LIN {X 0,Y 424.164,Z 335.01,A -85,B 0,C 180,E1 -10008.17,E2 -10008.17} C_VEL
LIN {X 0,Y 418.479,Z 320.385,A -85,B 0,C 180,E1 -10008.722,E2 -10008.722} C_VEL
LIN {X 0,Y 418.313,Z 319.478,A -85,B 0,C 180,E1 -10008.901,E2 -10008.901} C_VEL
LIN {X 0,Y 418.234,Z 319.369,A -85,B 0,C 180,E1 -10012.448,E2 -10012.448} C_VEL
LIN {X 0,Y 418.244,Z 319.388,A -85,B 0,C 180,E1 -10014.852,E2 -10014.852} C_VEL
LIN {X 0,Y 418.201,Z 319.366,A -85,B 0,C 180,E1 -10018.069,E2 -10018.069} C_VEL
LIN {X 0,Y 418.233,Z 319.388,A -85,B 0,C 180,E1 -10021.018,E2 -10021.018} C_VEL
LIN {X 0,Y 418.25,Z 319.387,A -85,B 0,C 180,E1 -10024.577,E2 -10024.577} C_VEL
LIN {X 0,Y 418.216,Z 319.377,A -85,B 0,C 180,E1 -10027.831,E2 -10027.831} C_VEL
LIN {X 0,Y 418.204,Z 319.389,A -85,B 0,C 180,E1 -10030.949,E2 -10030.949} C_VEL
LIN {X 0,Y 418.198,Z 319.375,A -85,B 0,C 180,E1 -10033.727,E2 -10033.727} C_VEL
LIN {X 0,Y 418.195,Z 319.394,A -85,B 0,C 180,E1 -10036.447,E2 -10036.447} C_VEL
LIN {X 0,Y 418.202,Z 319.379,A -85,B 0,C 180,E1 -10039.132,E2 -10039.132} C_VEL
LIN {X 0,Y 418.231,Z 319.378,A -85,B 0,C 180,E1 -10042.775,E2 -10042.775} C_VEL
LIN {X 0,Y 418.227,Z 319.39,A -85,B 0,C 180,E1 -10046.321,E2 -10046.321} C_VEL
LIN {X 0,Y 418.232,Z 319.36,A -85,B 0,C 180,E1 -10049.727,E2 -10049.727} C_VEL
LIN {X 0,Y 418.204,Z 319.382,A -85,B 0,C 180,E1 -10053.016,E2 -10053.016} C_VEL
LIN {X 0,Y 418.248,Z 319.387,A -85,B 0,C 180,E1 -10056.216,E2 -10056.216} C_VEL
LIN {X 0,Y 418.238,Z 319.376,A -85,B 0,C 180,E1 -10059.336,E2 -10059.336} C_VEL
LIN {X 0,Y 418.266,Z 319.387,A -85,B 0,C 180,E1 -10062.395,E2 -10062.395} C_VEL
LIN {X 0,Y 418.279,Z 319.367,A -85,B 0,C 180,E1 -10065.402,E2 -10065.402} C_VEL
LIN {X 0,Y 418.303,Z 319.381,A -85,B 0,C 180,E1 -10068.369,E2 -10068.369} C_VEL
LIN {X 0,Y 418.439,Z 319.353,A -85,B 0,C 180,E1 -10072.278,E2 -10072.278} C_VEL
LIN {X 0,Y 418.456,Z 319.357,A -85,B 0,C 180,E1 -10074.216,E2 -10074.216} C_VEL
LIN {X 0,Y 418.529,Z 319.347,A -85,B 0,C 180,E1 -10078.075,E2 -10078.075} C_VEL
LIN {X 0,Y 418.463,Z 319.355,A -85,B 0,C 180,E1 -10080.962,E2 -10080.962} C_VEL
LIN {X 0,Y 418.461,Z 319.357,A -85,B 0,C 180,E1 -10082.888,E2 -10082.888} C_VEL
LIN {X 0,Y 418.49,Z 319.346,A -85,B 0,C 180,E1 -10085.783,E2 -10085.783} C_VEL
LIN {X 0,Y 418.366,Z 319.37,A -85,B 0,C 180,E1 -10088.696,E2 -10088.696} C_VEL
LIN {X 0,Y 418.346,Z 319.364,A -85,B 0,C 180,E1 -10092.615,E2 -10092.615} C_VEL
LIN {X 0,Y 418.293,Z 319.377,A -85,B 0,C 180,E1 -10095.594,E2 -10095.594} C_VEL
LIN {X 0,Y 418.267,Z 319.373,A -85,B 0,C 180,E1 -10098.618,E2 -10098.618} C_VEL
LIN {X 0,Y 418.227,Z 319.371,A -85,B 0,C 180,E1 -10101.697,E2 -10101.697} C_VEL
LIN {X 0,Y 418.238,Z 319.385,A -85,B 0,C 180,E1 -10104.853,E2 -10104.853} C_VEL
LIN {X 0,Y 418.218,Z 319.377,A -85,B 0,C 180,E1 -10108.069,E2 -10108.069} C_VEL
LIN {X 0,Y 418.205,Z 319.389,A -85,B 0,C 180,E1 -10111.397,E2 -10111.397} C_VEL
LIN {X 0,Y 418.246,Z 319.377,A -85,B 0,C 180,E1 -10114.578,E2 -10114.578} C_VEL
LIN {X 0,Y 418.211,Z 319.392,A -85,B 0,C 180,E1 -10117.832,E2 -10117.832} C_VEL
LIN {X 0,Y 418.203,Z 319.39,A -85,B 0,C 180,E1 -10120.95,E2 -10120.95} C_VEL
LIN {X 0,Y 418.198,Z 319.378,A -85,B 0,C 180,E1 -10123.729,E2 -10123.729} C_VEL
LIN {X 0,Y 418.194,Z 319.382,A -85,B 0,C 180,E1 -10126.448,E2 -10126.448} C_VEL
LIN {X 0,Y 418.203,Z 319.387,A -85,B 0,C 180,E1 -10129.134,E2 -10129.134} C_VEL
LIN {X 0,Y 418.23,Z 319.388,A -85,B 0,C 180,E1 -10132.776,E2 -10132.776} C_VEL
LIN {X 0,Y 418.23,Z 319.385,A -85,B 0,C 180,E1 -10136.322,E2 -10136.322} C_VEL
LIN {X 0,Y 418.282,Z 319.584,A -85,B 0,C 180,E1 -10137.85,E2 -10137.85} C_VEL
LIN {X 0,Y 421.611,Z 333.785,A -85,B 0,C 180,E1 -10140.357,E2 -10140.357} C_VEL
LIN {X 0,Y 422.933,Z 341.038,A -85,B 0,C 180,E1 -10141.57,E2 -10141.57} C_VEL
LIN {X 0,Y 421.685,Z 360.969,A -85,B 0,C 180,E1 -10144.586,E2 -10144.586} C_VEL
LIN {X 0,Y 420.463,Z 381.404,A -85,B 0,C 180,E1 -10147.65,E2 -10147.65} C_VEL
LIN {X 0,Y 419.398,Z 403.02,A -85,B 0,C 180,E1 -10150.874,E2 -10150.874} C_VEL
LIN {X 0,Y 423.294,Z 439.321,A -85,B 0,C 180,E1 -10151.702,E2 -10151.702} C_VEL
LIN {X 0,Y 422.516,Z 513.567,A -85,B 0,C 180,E1 -10152.984,E2 -10152.984} C_VEL
LIN {X 0,Y 422.025,Z 526.877,A -85,B 0,C 180,E1 -10153.399,E2 -10153.399} C_VEL
LIN {X 0,Y 421.283,Z 539.091,A -85,B 0,C 180,E1 -10153.961,E2 -10153.961} C_VEL
LIN {X 0,Y 420.463,Z 551.46,A -85,B 0,C 180,E1 -10154.737,E2 -10154.737} C_VEL
LIN {X 0,Y 419.557,Z 563.169,A -85,B 0,C 180,E1 -10155.696,E2 -10155.696} C_VEL
LIN {X 0,Y 418.897,Z 574.07,A -85,B 0,C 180,E1 -10156.82,E2 -10156.82} C_VEL
LIN {X 0,Y 418.543,Z 580.651,A -85,B 0,C 180,E1 -10157.638,E2 -10157.638} C_VEL
LIN {X 0,Y 417.995,Z 588.983,A -85,B 0,C 180,E1 -10158.851,E2 -10158.851} C_VEL
LIN {X 0,Y 417.634,Z 597.2,A -85,B 0,C 180,E1 -10160.312,E2 -10160.312} C_VEL
LIN {X 0,Y 417.519,Z 603.829,A -85,B 0,C 180,E1 -10161.774,E2 -10161.774} C_VEL
LIN {X 0,Y 417.47,Z 609.435,A -85,B 0,C 180,E1 -10163.34,E2 -10163.34} C_VEL
LIN {X 0,Y 417.644,Z 614.342,A -85,B 0,C 180,E1 -10165.174,E2 -10165.174} C_VEL
LIN {X 0,Y 417.711,Z 616.278,A -85,B 0,C 180,E1 -10166.141,E2 -10166.141} C_VEL
LIN {X 0,Y 417.687,Z 617.72,A -85,B 0,C 180,E1 -10167.107,E2 -10167.107} C_VEL
LIN {X 0,Y 417.947,Z 619.416,A -85,B 0,C 180,E1 -10169.037,E2 -10169.037} C_VEL
LIN {X 0,Y 417.96,Z 619.641,A -85,B 0,C 180,E1 -10170,E2 -10170} C_VEL
LIN {X 0,Y 417.947,Z 619.415,A -85,B 0,C 180,E1 -10170.963,E2 -10170.963} C_VEL
LIN {X 0,Y 417.688,Z 617.719,A -85,B 0,C 180,E1 -10172.893,E2 -10172.893} C_VEL
LIN {X 0,Y 417.711,Z 616.275,A -85,B 0,C 180,E1 -10173.859,E2 -10173.859} C_VEL
LIN {X 0,Y 417.551,Z 613.215,A -85,B 0,C 180,E1 -10175.312,E2 -10175.312} C_VEL
LIN {X 0,Y 417.519,Z 609.099,A -85,B 0,C 180,E1 -10176.767,E2 -10176.767} C_VEL
LIN {X 0,Y 417.519,Z 602.781,A -85,B 0,C 180,E1 -10178.47,E2 -10178.47} C_VEL
LIN {X 0,Y 417.664,Z 595.91,A -85,B 0,C 180,E1 -10179.932,E2 -10179.932} C_VEL
LIN {X 0,Y 418.089,Z 587.435,A -85,B 0,C 180,E1 -10181.391,E2 -10181.391} C_VEL
LIN {X 0,Y 418.703,Z 578.787,A -85,B 0,C 180,E1 -10182.604,E2 -10182.604} C_VEL
LIN {X 0,Y 419.221,Z 569.303,A -85,B 0,C 180,E1 -10183.697,E2 -10183.697} C_VEL
LIN {X 0,Y 419.925,Z 557.585,A -85,B 0,C 180,E1 -10184.787,E2 -10184.787} C_VEL
LIN {X 0,Y 420.82,Z 546.111,A -85,B 0,C 180,E1 -10185.622,E2 -10185.622} C_VEL
LIN {X 0,Y 421.537,Z 534.336,A -85,B 0,C 180,E1 -10186.278,E2 -10186.278} C_VEL
LIN {X 0,Y 422.248,Z 521.736,A -85,B 0,C 180,E1 -10186.778,E2 -10186.778} C_VEL
LIN {X 0,Y 422.652,Z 508.962,A -85,B 0,C 180,E1 -10187.104,E2 -10187.104} C_VEL
LIN {X 0,Y 423.252,Z 438.649,A -85,B 0,C 180,E1 -10188.305,E2 -10188.305} C_VEL
LIN {X 0,Y 419.395,Z 403.264,A -85,B 0,C 180,E1 -10189.104,E2 -10189.104} C_VEL
LIN {X 0,Y 419.602,Z 397.115,A -85,B 0,C 180,E1 -10189.982,E2 -10189.982} C_VEL
LIN {X 0,Y 420.761,Z 376.002,A -85,B 0,C 180,E1 -10193.15,E2 -10193.15} C_VEL
LIN {X 0,Y 422.195,Z 352.327,A -85,B 0,C 180,E1 -10196.708,E2 -10196.708} C_VEL
LIN {X 0,Y 422.873,Z 340.757,A -85,B 0,C 180,E1 -10198.467,E2 -10198.467} C_VEL
LIN {X 0,Y 420.636,Z 329.564,A -85,B 0,C 180,E1 -10200.358,E2 -10200.358} C_VEL
LIN {X 0,Y 418.275,Z 319.506,A -85,B 0,C 180,E1 -10202.169,E2 -10202.169} C_VEL
LIN {X 0,Y 418.247,Z 319.383,A -85,B 0,C 180,E1 -10204.841,E2 -10204.841} C_VEL
LIN {X 0,Y 418.231,Z 319.382,A -85,B 0,C 180,E1 -10208.443,E2 -10208.443} C_VEL
LIN {X 0,Y 418.215,Z 319.392,A -85,B 0,C 180,E1 -10212.235,E2 -10212.235} C_VEL
LIN {X 0,Y 418.23,Z 319.362,A -85,B 0,C 180,E1 -10215.108,E2 -10215.108} C_VEL
LIN {X 0,Y 418.216,Z 319.389,A -85,B 0,C 180,E1 -10217.764,E2 -10217.764} C_VEL
LIN {X 0,Y 418.228,Z 319.36,A -85,B 0,C 180,E1 -10221.555,E2 -10221.555} C_VEL
LIN {X 0,Y 418.244,Z 319.368,A -85,B 0,C 180,E1 -10225.157,E2 -10225.157} C_VEL
LIN {X 0,Y 418.238,Z 319.385,A -85,B 0,C 180,E1 -10227.471,E2 -10227.471} C_VEL
LIN {X 0,Y 418.257,Z 319.372,A -85,B 0,C 180,E1 -10230.896,E2 -10230.896} C_VEL
LIN {X 0,Y 418.224,Z 319.391,A -85,B 0,C 180,E1 -10234.093,E2 -10234.093} C_VEL
LIN {X 0,Y 418.221,Z 319.384,A -85,B 0,C 180,E1 -10237.263,E2 -10237.263} C_VEL
LIN {X 0,Y 418.276,Z 319.371,A -85,B 0,C 180,E1 -10240.364,E2 -10240.364} C_VEL
LIN {X 0,Y 418.309,Z 319.377,A -85,B 0,C 180,E1 -10243.404,E2 -10243.404} C_VEL
LIN {X 0,Y 418.339,Z 319.362,A -85,B 0,C 180,E1 -10246.999,E2 -10246.999} C_VEL
LIN {X 0,Y 418.327,Z 319.374,A -85,B 0,C 180,E1 -10250.328,E2 -10250.328} C_VEL
LIN {X 0,Y 418.458,Z 319.353,A -85,B 0,C 180,E1 -10253.248,E2 -10253.248} C_VEL
LIN {X 0,Y 418.313,Z 319.369,A -85,B 0,C 180,E1 -10255.181,E2 -10255.181} C_VEL
LIN {X 0,Y 418.524,Z 319.349,A -85,B 0,C 180,E1 -10258.075,E2 -10258.075} C_VEL
LIN {X 0,Y 418.398,Z 319.353,A -85,B 0,C 180,E1 -10260.963,E2 -10260.963} C_VEL
LIN {X 0,Y 418.473,Z 319.352,A -85,B 0,C 180,E1 -10262.888,E2 -10262.888} C_VEL
LIN {X 0,Y 418.434,Z 319.354,A -85,B 0,C 180,E1 -10266.752,E2 -10266.752} C_VEL
LIN {X 0,Y 418.329,Z 319.373,A -85,B 0,C 180,E1 -10269.672,E2 -10269.672} C_VEL
LIN {X 0,Y 418.339,Z 319.37,A -85,B 0,C 180,E1 -10273.001,E2 -10273.001} C_VEL
LIN {X 0,Y 418.304,Z 319.374,A -85,B 0,C 180,E1 -10276.735,E2 -10276.735} C_VEL
LIN {X 0,Y 418.263,Z 319.377,A -85,B 0,C 180,E1 -10279.79,E2 -10279.79} C_VEL
LIN {X 0,Y 418.221,Z 319.384,A -85,B 0,C 180,E1 -10282.737,E2 -10282.737} C_VEL
LIN {X 0,Y 418.212,Z 319.383,A -85,B 0,C 180,E1 -10285.908,E2 -10285.908} C_VEL
LIN {X 0,Y 418.25,Z 319.355,A -85,B 0,C 180,E1 -10289.163,E2 -10289.163} C_VEL
LIN {X 0,Y 418.246,Z 319.378,A -85,B 0,C 180,E1 -10292.843,E2 -10292.843} C_VEL
LIN {X 0,Y 418.238,Z 319.381,A -85,B 0,C 180,E1 -10296.238,E2 -10296.238} C_VEL
LIN {X 0,Y 418.194,Z 319.371,A -85,B 0,C 180,E1 -10299.689,E2 -10299.689} C_VEL
LIN {X 0,Y 418.203,Z 319.388,A -85,B 0,C 180,E1 -10302.318,E2 -10302.318} C_VEL
LIN {X 0,Y 418.232,Z 319.384,A -85,B 0,C 180,E1 -10305.109,E2 -10305.109} C_VEL
LIN {X 0,Y 418.214,Z 319.379,A -85,B 0,C 180,E1 -10307.765,E2 -10307.765} C_VEL
LIN {X 0,Y 418.233,Z 319.38,A -85,B 0,C 180,E1 -10311.557,E2 -10311.557} C_VEL
LIN {X 0,Y 418.249,Z 319.388,A -85,B 0,C 180,E1 -10315.159,E2 -10315.159} C_VEL
LIN {X 0,Y 418.237,Z 319.38,A -85,B 0,C 180,E1 -10317.472,E2 -10317.472} C_VEL
LIN {X 0,Y 418.258,Z 319.376,A -85,B 0,C 180,E1 -10320.899,E2 -10320.899} C_VEL
LIN {X 0,Y 418.21,Z 319.379,A -85,B 0,C 180,E1 -10324.092,E2 -10324.092} C_VEL
LIN {X 0,Y 418.227,Z 319.373,A -85,B 0,C 180,E1 -10327.264,E2 -10327.264} C_VEL
LIN {X 0,Y 418.312,Z 319.345,A -85,B 0,C 180,E1 -10330.876,E2 -10330.876} C_VEL
LIN {X 0,Y 418.37,Z 319.77,A -85,B 0,C 180,E1 -10331.292,E2 -10331.292} C_VEL
LIN {X 0,Y 418.751,Z 321.14,A -85,B 0,C 180,E1 -10331.419,E2 -10331.419} C_VEL
LIN {X 0,Y 424.249,Z 335.165,A -85,B 0,C 180,E1 -10331.934,E2 -10331.934} C_VEL
LIN {X 0,Y 423.684,Z 400.146,A -85,B 0,C 180,E1 -10333.063,E2 -10333.063} C_VEL
LIN {X 0,Y 423.564,Z 412.838,A -85,B 0,C 180,E1 -10333.461,E2 -10333.461} C_VEL
LIN {X 0,Y 423.267,Z 425.198,A -85,B 0,C 180,E1 -10334.038,E2 -10334.038} C_VEL
LIN {X 0,Y 422.856,Z 437.548,A -85,B 0,C 180,E1 -10334.824,E2 -10334.824} C_VEL
LIN {X 0,Y 422.141,Z 449.13,A -85,B 0,C 180,E1 -10335.785,E2 -10335.785} C_VEL
LIN {X 0,Y 421.492,Z 459.468,A -85,B 0,C 180,E1 -10336.869,E2 -10336.869} C_VEL
LIN {X 0,Y 420.95,Z 467.894,A -85,B 0,C 180,E1 -10337.954,E2 -10337.954} C_VEL
LIN {X 0,Y 420.346,Z 475.653,A -85,B 0,C 180,E1 -10339.159,E2 -10339.159} C_VEL
LIN {X 0,Y 419.765,Z 483.331,A -85,B 0,C 180,E1 -10340.629,E2 -10340.629} C_VEL
LIN {X 0,Y 419.323,Z 489.087,A -85,B 0,C 180,E1 -10342.002,E2 -10342.002} C_VEL
LIN {X 0,Y 419.063,Z 493.36,A -85,B 0,C 180,E1 -10343.258,E2 -10343.258} C_VEL
LIN {X 0,Y 418.611,Z 497.256,A -85,B 0,C 180,E1 -10344.702,E2 -10344.702} C_VEL
LIN {X 0,Y 418.384,Z 499.239,A -85,B 0,C 180,E1 -10345.678,E2 -10345.678} C_VEL
LIN {X 0,Y 417.623,Z 500.71,A -85,B 0,C 180,E1 -10346.457,E2 -10346.457} C_VEL
LIN {X 0,Y 414.712,Z 502.691,A -85,B 0,C 180,E1 -10347.733,E2 -10347.733} C_VEL
LIN {X 0,Y 412.317,Z 503.759,A -85,B 0,C 180,E1 -10348.773,E2 -10348.773} C_VEL
LIN {X 0,Y 411.309,Z 504.179,A -85,B 0,C 180,E1 -10349.583,E2 -10349.583} C_VEL
LIN {X 0,Y 411.235,Z 504.22,A -85,B 0,C 180,E1 -10349.857,E2 -10349.857} C_VEL
LIN {X 0,Y 411.257,Z 504.07,A -85,B 0,C 180,E1 -10350.979,E2 -10350.979} C_VEL
LIN {X 0,Y 411.181,Z 503.516,A -85,B 0,C 180,E1 -10351.959,E2 -10351.959} C_VEL
LIN {X 0,Y 411.332,Z 502.561,A -85,B 0,C 180,E1 -10352.938,E2 -10352.938} C_VEL
LIN {X 0,Y 411.294,Z 501.258,A -85,B 0,C 180,E1 -10353.919,E2 -10353.919} C_VEL
LIN {X 0,Y 411.607,Z 498.444,A -85,B 0,C 180,E1 -10355.388,E2 -10355.388} C_VEL
LIN {X 0,Y 412.065,Z 494.62,A -85,B 0,C 180,E1 -10356.857,E2 -10356.857} C_VEL
LIN {X 0,Y 412.366,Z 489.544,A -85,B 0,C 180,E1 -10358.379,E2 -10358.379} C_VEL
LIN {X 0,Y 413.052,Z 482.312,A -85,B 0,C 180,E1 -10360.044,E2 -10360.044} C_VEL
LIN {X 0,Y 413.751,Z 474.285,A -85,B 0,C 180,E1 -10361.513,E2 -10361.513} C_VEL
LIN {X 0,Y 414.321,Z 466.066,A -85,B 0,C 180,E1 -10362.739,E2 -10362.739} C_VEL
LIN {X 0,Y 414.933,Z 457.038,A -85,B 0,C 180,E1 -10363.842,E2 -10363.842} C_VEL
LIN {X 0,Y 415.695,Z 446.536,A -85,B 0,C 180,E1 -10364.872,E2 -10364.872} C_VEL
LIN {X 0,Y 416.207,Z 434.882,A -85,B 0,C 180,E1 -10365.787,E2 -10365.787} C_VEL
LIN {X 0,Y 416.655,Z 423.452,A -85,B 0,C 180,E1 -10366.474,E2 -10366.474} C_VEL
LIN {X 0,Y 416.858,Z 410.602,A -85,B 0,C 180,E1 -10367.033,E2 -10367.033} C_VEL
LIN {X 0,Y 416.904,Z 396.844,A -85,B 0,C 180,E1 -10367.411,E2 -10367.411} C_VEL
LIN {X 0,Y 417.432,Z 336.493,A -85,B 0,C 180,E1 -10368.464,E2 -10368.464} C_VEL
LIN {X 0,Y 411.427,Z 321.136,A -85,B 0,C 180,E1 -10369.068,E2 -10369.068} C_VEL
LIN {X 0,Y 411.278,Z 320.312,A -85,B 0,C 180,E1 -10369.27,E2 -10369.27} C_VEL
LIN {X 0,Y 411.187,Z 320.251,A -85,B 0,C 180,E1 -10373.148,E2 -10373.148} C_VEL
LIN {X 0,Y 411.163,Z 320.246,A -85,B 0,C 180,E1 -10376.386,E2 -10376.386} C_VEL
LIN {X 0,Y 411.193,Z 320.261,A -85,B 0,C 180,E1 -10379.713,E2 -10379.713} C_VEL
LIN {X 0,Y 411.201,Z 320.258,A -85,B 0,C 180,E1 -10383.156,E2 -10383.156} C_VEL
LIN {X 0,Y 411.188,Z 320.257,A -85,B 0,C 180,E1 -10386.551,E2 -10386.551} C_VEL
LIN {X 0,Y 411.166,Z 320.266,A -85,B 0,C 180,E1 -10389.719,E2 -10389.719} C_VEL
LIN {X 0,Y 411.158,Z 320.251,A -85,B 0,C 180,E1 -10393.135,E2 -10393.135} C_VEL
LIN {X 0,Y 411.16,Z 320.266,A -85,B 0,C 180,E1 -10395.881,E2 -10395.881} C_VEL
LIN {X 0,Y 411.153,Z 320.255,A -85,B 0,C 180,E1 -10399.492,E2 -10399.492} C_VEL
LIN {X 0,Y 411.179,Z 320.246,A -85,B 0,C 180,E1 -10402.024,E2 -10402.024} C_VEL
LIN {X 0,Y 411.197,Z 320.263,A -85,B 0,C 180,E1 -10405.123,E2 -10405.123} C_VEL
LIN {X 0,Y 411.158,Z 320.26,A -85,B 0,C 180,E1 -10408.002,E2 -10408.002} C_VEL
LIN {X 0,Y 411.165,Z 320.241,A -85,B 0,C 180,E1 -10411.406,E2 -10411.406} C_VEL
LIN {X 0,Y 411.182,Z 320.266,A -85,B 0,C 180,E1 -10414.941,E2 -10414.941} C_VEL
LIN {X 0,Y 411.194,Z 320.26,A -85,B 0,C 180,E1 -10417.913,E2 -10417.913} C_VEL
LIN {X 0,Y 411.21,Z 320.261,A -85,B 0,C 180,E1 -10421.051,E2 -10421.051} C_VEL
LIN {X 0,Y 411.236,Z 320.257,A -85,B 0,C 180,E1 -10424.131,E2 -10424.131} C_VEL
LIN {X 0,Y 411.296,Z 320.247,A -85,B 0,C 180,E1 -10427.165,E2 -10427.165} C_VEL
LIN {X 0,Y 411.273,Z 320.255,A -85,B 0,C 180,E1 -10430.161,E2 -10430.161} C_VEL
LIN {X 0,Y 411.378,Z 320.234,A -85,B 0,C 180,E1 -10433.132,E2 -10433.132} C_VEL
LIN {X 0,Y 411.28,Z 320.252,A -85,B 0,C 180,E1 -10435.099,E2 -10435.099} C_VEL
LIN {X 0,Y 411.498,Z 320.223,A -85,B 0,C 180,E1 -10438.042,E2 -10438.042} C_VEL
LIN {X 0,Y 411.493,Z 320.225,A -85,B 0,C 180,E1 -10441.957,E2 -10441.957} C_VEL
LIN {X 0,Y 411.436,Z 320.225,A -85,B 0,C 180,E1 -10445.883,E2 -10445.883} C_VEL
LIN {X 0,Y 411.406,Z 320.232,A -85,B 0,C 180,E1 -10447.855,E2 -10447.855} C_VEL
LIN {X 0,Y 411.266,Z 320.251,A -85,B 0,C 180,E1 -10451.833,E2 -10451.833} C_VEL
LIN {X 0,Y 411.251,Z 320.255,A -85,B 0,C 180,E1 -10454.853,E2 -10454.853} C_VEL
LIN {X 0,Y 411.237,Z 320.259,A -85,B 0,C 180,E1 -10457.916,E2 -10457.916} C_VEL
LIN {X 0,Y 411.189,Z 320.246,A -85,B 0,C 180,E1 -10461.035,E2 -10461.035} C_VEL
LIN {X 0,Y 411.186,Z 320.268,A -85,B 0,C 180,E1 -10464.218,E2 -10464.218} C_VEL
LIN {X 0,Y 411.175,Z 320.258,A -85,B 0,C 180,E1 -10467.484,E2 -10467.484} C_VEL
LIN {X 0,Y 411.192,Z 320.255,A -85,B 0,C 180,E1 -10469.713,E2 -10469.713} C_VEL
LIN {X 0,Y 411.199,Z 320.259,A -85,B 0,C 180,E1 -10473.157,E2 -10473.157} C_VEL
LIN {X 0,Y 411.183,Z 320.266,A -85,B 0,C 180,E1 -10476.552,E2 -10476.552} C_VEL
LIN {X 0,Y 411.163,Z 320.261,A -85,B 0,C 180,E1 -10479.721,E2 -10479.721} C_VEL
LIN {X 0,Y 411.159,Z 320.262,A -85,B 0,C 180,E1 -10483.136,E2 -10483.136} C_VEL
LIN {X 0,Y 411.158,Z 320.248,A -85,B 0,C 180,E1 -10485.883,E2 -10485.883} C_VEL
LIN {X 0,Y 411.143,Z 320.267,A -85,B 0,C 180,E1 -10488.775,E2 -10488.775} C_VEL
LIN {X 0,Y 411.178,Z 320.266,A -85,B 0,C 180,E1 -10492.025,E2 -10492.025} C_VEL
LIN {X 0,Y 411.199,Z 320.259,A -85,B 0,C 180,E1 -10495.124,E2 -10495.124} C_VEL
LIN {X 0,Y 411.231,Z 320.494,A -85,B 0,C 180,E1 -10497.539,E2 -10497.539} C_VEL
LIN {X 0,Y 414.675,Z 335.185,A -85,B 0,C 180,E1 -10500.187,E2 -10500.187} C_VEL
LIN {X 0,Y 416.05,Z 342.591,A -85,B 0,C 180,E1 -10501.45,E2 -10501.45} C_VEL
LIN {X 0,Y 414.782,Z 361.752,A -85,B 0,C 180,E1 -10504.402,E2 -10504.402} C_VEL
LIN {X 0,Y 413.494,Z 382.134,A -85,B 0,C 180,E1 -10507.517,E2 -10507.517} C_VEL
LIN {X 0,Y 412.436,Z 401.9,A -85,B 0,C 180,E1 -10510.529,E2 -10510.529} C_VEL
LIN {X 0,Y 415.827,Z 433.041,A -85,B 0,C 180,E1 -10511.269,E2 -10511.269} C_VEL
LIN {X 0,Y 416.533,Z 441.796,A -85,B 0,C 180,E1 -10511.456,E2 -10511.456} C_VEL
LIN {X 0,Y 415.691,Z 512.586,A -85,B 0,C 180,E1 -10512.696,E2 -10512.696} C_VEL
LIN {X 0,Y 415.186,Z 525.891,A -85,B 0,C 180,E1 -10513.118,E2 -10513.118} C_VEL
LIN {X 0,Y 414.433,Z 538.104,A -85,B 0,C 180,E1 -10513.688,E2 -10513.688} C_VEL
LIN {X 0,Y 413.726,Z 548.767,A -85,B 0,C 180,E1 -10514.356,E2 -10514.356} C_VEL
LIN {X 0,Y 412.815,Z 559.534,A -85,B 0,C 180,E1 -10515.205,E2 -10515.205} C_VEL
LIN {X 0,Y 412.178,Z 569.513,A -85,B 0,C 180,E1 -10516.19,E2 -10516.19} C_VEL
LIN {X 0,Y 411.592,Z 579.662,A -85,B 0,C 180,E1 -10517.426,E2 -10517.426} C_VEL
LIN {X 0,Y 410.97,Z 587.989,A -85,B 0,C 180,E1 -10518.658,E2 -10518.658} C_VEL
LIN {X 0,Y 410.555,Z 596.202,A -85,B 0,C 180,E1 -10520.144,E2 -10520.144} C_VEL
LIN {X 0,Y 410.441,Z 602.835,A -85,B 0,C 180,E1 -10521.631,E2 -10521.631} C_VEL
LIN {X 0,Y 410.419,Z 608.703,A -85,B 0,C 180,E1 -10523.31,E2 -10523.31} C_VEL
LIN {X 0,Y 410.567,Z 613.354,A -85,B 0,C 180,E1 -10525.09,E2 -10525.09} C_VEL
LIN {X 0,Y 410.669,Z 615.296,A -85,B 0,C 180,E1 -10526.075,E2 -10526.075} C_VEL
LIN {X 0,Y 410.642,Z 616.738,A -85,B 0,C 180,E1 -10527.057,E2 -10527.057} C_VEL
LIN {X 0,Y 410.918,Z 618.438,A -85,B 0,C 180,E1 -10529.02,E2 -10529.02} C_VEL
LIN {X 0,Y 410.935,Z 618.663,A -85,B 0,C 180,E1 -10530,E2 -10530} C_VEL
LIN {X 0,Y 410.918,Z 618.436,A -85,B 0,C 180,E1 -10530.98,E2 -10530.98} C_VEL
LIN {X 0,Y 410.642,Z 616.737,A -85,B 0,C 180,E1 -10532.943,E2 -10532.943} C_VEL
LIN {X 0,Y 410.67,Z 615.292,A -85,B 0,C 180,E1 -10533.925,E2 -10533.925} C_VEL
LIN {X 0,Y 410.48,Z 612.226,A -85,B 0,C 180,E1 -10535.403,E2 -10535.403} C_VEL
LIN {X 0,Y 410.434,Z 608.105,A -85,B 0,C 180,E1 -10536.884,E2 -10536.884} C_VEL
LIN {X 0,Y 410.451,Z 601.785,A -85,B 0,C 180,E1 -10538.616,E2 -10538.616} C_VEL
LIN {X 0,Y 410.609,Z 594.911,A -85,B 0,C 180,E1 -10540.104,E2 -10540.104} C_VEL
LIN {X 0,Y 411.046,Z 586.433,A -85,B 0,C 180,E1 -10541.589,E2 -10541.589} C_VEL
LIN {X 0,Y 411.701,Z 577.786,A -85,B 0,C 180,E1 -10542.821,E2 -10542.821} C_VEL
LIN {X 0,Y 412.347,Z 567.111,A -85,B 0,C 180,E1 -10544.056,E2 -10544.056} C_VEL
LIN {X 0,Y 413.032,Z 556.589,A -85,B 0,C 180,E1 -10545.039,E2 -10545.039} C_VEL
LIN {X 0,Y 413.927,Z 545.11,A -85,B 0,C 180,E1 -10545.889,E2 -10545.889} C_VEL
LIN {X 0,Y 414.729,Z 533.341,A -85,B 0,C 180,E1 -10546.553,E2 -10546.553} C_VEL
LIN {X 0,Y 415.483,Z 519.818,A -85,B 0,C 180,E1 -10547.091,E2 -10547.091} C_VEL
LIN {X 0,Y 415.838,Z 506.408,A -85,B 0,C 180,E1 -10547.425,E2 -10547.425} C_VEL
LIN {X 0,Y 416.42,Z 438.976,A -85,B 0,C 180,E1 -10548.592,E2 -10548.592} C_VEL
LIN {X 0,Y 412.45,Z 402.247,A -85,B 0,C 180,E1 -10549.438,E2 -10549.438} C_VEL
LIN {X 0,Y 412.825,Z 393.906,A -85,B 0,C 180,E1 -10550.672,E2 -10550.672} C_VEL
LIN {X 0,Y 414.078,Z 371.9,A -85,B 0,C 180,E1 -10554.038,E2 -10554.038} C_VEL
LIN {X 0,Y 415.439,Z 351.412,A -85,B 0,C 180,E1 -10557.178,E2 -10557.178} C_VEL
LIN {X 0,Y 415.988,Z 342.084,A -85,B 0,C 180,E1 -10558.625,E2 -10558.625} C_VEL
LIN {X 0,Y 413.593,Z 330.359,A -85,B 0,C 180,E1 -10560.648,E2 -10560.648} C_VEL
LIN {X 0,Y 411.235,Z 320.374,A -85,B 0,C 180,E1 -10562.497,E2 -10562.497} C_VEL
LIN {X 0,Y 411.173,Z 320.258,A -85,B 0,C 180,E1 -10565.53,E2 -10565.53} C_VEL
LIN {X 0,Y 411.174,Z 320.254,A -85,B 0,C 180,E1 -10569.228,E2 -10569.228} C_VEL
LIN {X 0,Y 411.162,Z 320.266,A -85,B 0,C 180,E1 -10572.693,E2 -10572.693} C_VEL
LIN {X 0,Y 411.159,Z 320.248,A -85,B 0,C 180,E1 -10575.881,E2 -10575.881} C_VEL
LIN {X 0,Y 411.143,Z 320.27,A -85,B 0,C 180,E1 -10578.774,E2 -10578.774} C_VEL
LIN {X 0,Y 411.176,Z 320.228,A -85,B 0,C 180,E1 -10582.024,E2 -10582.024} C_VEL
LIN {X 0,Y 411.196,Z 320.245,A -85,B 0,C 180,E1 -10585.123,E2 -10585.123} C_VEL
LIN {X 0,Y 411.158,Z 320.272,A -85,B 0,C 180,E1 -10588.002,E2 -10588.002} C_VEL
LIN {X 0,Y 411.187,Z 320.252,A -85,B 0,C 180,E1 -10591.407,E2 -10591.407} C_VEL
LIN {X 0,Y 411.206,Z 320.261,A -85,B 0,C 180,E1 -10594.933,E2 -10594.933} C_VEL
LIN {X 0,Y 411.197,Z 320.25,A -85,B 0,C 180,E1 -10597.913,E2 -10597.913} C_VEL
LIN {X 0,Y 411.215,Z 320.249,A -85,B 0,C 180,E1 -10601.051,E2 -10601.051} C_VEL
LIN {X 0,Y 411.246,Z 320.257,A -85,B 0,C 180,E1 -10604.131,E2 -10604.131} C_VEL
LIN {X 0,Y 411.296,Z 320.24,A -85,B 0,C 180,E1 -10607.165,E2 -10607.165} C_VEL
LIN {X 0,Y 411.28,Z 320.254,A -85,B 0,C 180,E1 -10610.161,E2 -10610.161} C_VEL
LIN {X 0,Y 411.424,Z 320.228,A -85,B 0,C 180,E1 -10613.132,E2 -10613.132} C_VEL
LIN {X 0,Y 411.286,Z 320.244,A -85,B 0,C 180,E1 -10615.099,E2 -10615.099} C_VEL
LIN {X 0,Y 411.493,Z 320.226,A -85,B 0,C 180,E1 -10618.043,E2 -10618.043} C_VEL
LIN {X 0,Y 411.369,Z 320.228,A -85,B 0,C 180,E1 -10620.979,E2 -10620.979} C_VEL
LIN {X 0,Y 411.431,Z 320.229,A -85,B 0,C 180,E1 -10622.937,E2 -10622.937} C_VEL
LIN {X 0,Y 411.383,Z 320.232,A -85,B 0,C 180,E1 -10626.868,E2 -10626.868} C_VEL
LIN {X 0,Y 411.282,Z 320.254,A -85,B 0,C 180,E1 -10629.839,E2 -10629.839} C_VEL
LIN {X 0,Y 411.299,Z 320.247,A -85,B 0,C 180,E1 -10633.104,E2 -10633.104} C_VEL
LIN {X 0,Y 411.251,Z 320.253,A -85,B 0,C 180,E1 -10636.889,E2 -10636.889} C_VEL
LIN {X 0,Y 411.225,Z 320.252,A -85,B 0,C 180,E1 -10639.987,E2 -10639.987} C_VEL
LIN {X 0,Y 411.182,Z 320.263,A -85,B 0,C 180,E1 -10643.149,E2 -10643.149} C_VEL
LIN {X 0,Y 411.165,Z 320.258,A -85,B 0,C 180,E1 -10646.386,E2 -10646.386} C_VEL
LIN {X 0,Y 411.189,Z 320.232,A -85,B 0,C 180,E1 -10649.714,E2 -10649.714} C_VEL
LIN {X 0,Y 411.199,Z 320.258,A -85,B 0,C 180,E1 -10653.157,E2 -10653.157} C_VEL
LIN {X 0,Y 411.186,Z 320.259,A -85,B 0,C 180,E1 -10656.553,E2 -10656.553} C_VEL
LIN {X 0,Y 411.163,Z 320.246,A -85,B 0,C 180,E1 -10659.721,E2 -10659.721} C_VEL
LIN {X 0,Y 411.159,Z 320.27,A -85,B 0,C 180,E1 -10663.136,E2 -10663.136} C_VEL
LIN {X 0,Y 411.16,Z 320.253,A -85,B 0,C 180,E1 -10665.883,E2 -10665.883} C_VEL
LIN {X 0,Y 411.155,Z 320.272,A -85,B 0,C 180,E1 -10669.494,E2 -10669.494} C_VEL
LIN {X 0,Y 411.18,Z 320.254,A -85,B 0,C 180,E1 -10672.026,E2 -10672.026} C_VEL
LIN {X 0,Y 411.201,Z 320.265,A -85,B 0,C 180,E1 -10675.124,E2 -10675.124} C_VEL
LIN {X 0,Y 411.158,Z 320.264,A -85,B 0,C 180,E1 -10678.003,E2 -10678.003} C_VEL
LIN {X 0,Y 411.168,Z 320.249,A -85,B 0,C 180,E1 -10681.407,E2 -10681.407} C_VEL
LIN {X 0,Y 411.187,Z 320.266,A -85,B 0,C 180,E1 -10684.942,E2 -10684.942} C_VEL
LIN {X 0,Y 411.203,Z 320.246,A -85,B 0,C 180,E1 -10687.914,E2 -10687.914} C_VEL
LIN {X 0,Y 411.298,Z 320.359,A -85,B 0,C 180,E1 -10690.861,E2 -10690.861} C_VEL
LIN {X 0,Y 411.44,Z 321.123,A -85,B 0,C 180,E1 -10691.03,E2 -10691.03} C_VEL
LIN {X 0,Y 417.409,Z 336.438,A -85,B 0,C 180,E1 -10691.632,E2 -10691.632} C_VEL
LIN {X 0,Y 416.955,Z 401.145,A -85,B 0,C 180,E1 -10692.781,E2 -10692.781} C_VEL
LIN {X 0,Y 416.815,Z 413.829,A -85,B 0,C 180,E1 -10693.186,E2 -10693.186} C_VEL
LIN {X 0,Y 416.511,Z 426.184,A -85,B 0,C 180,E1 -10693.772,E2 -10693.772} C_VEL
LIN {X 0,Y 416.078,Z 438.531,A -85,B 0,C 180,E1 -10694.57,E2 -10694.57} C_VEL
LIN {X 0,Y 415.329,Z 450.113,A -85,B 0,C 180,E1 -10695.547,E2 -10695.547} C_VEL
LIN {X 0,Y 414.649,Z 460.45,A -85,B 0,C 180,E1 -10696.648,E2 -10696.648} C_VEL
LIN {X 0,Y 414.078,Z 468.876,A -85,B 0,C 180,E1 -10697.751,E2 -10697.751} C_VEL
LIN {X 0,Y 413.445,Z 476.633,A -85,B 0,C 180,E1 -10698.975,E2 -10698.975} C_VEL
LIN {X 0,Y 412.833,Z 484.311,A -85,B 0,C 180,E1 -10700.471,E2 -10700.471} C_VEL
LIN {X 0,Y 412.365,Z 490.067,A -85,B 0,C 180,E1 -10701.867,E2 -10701.867} C_VEL
LIN {X 0,Y 412.086,Z 494.339,A -85,B 0,C 180,E1 -10703.144,E2 -10703.144} C_VEL
LIN {X 0,Y 411.612,Z 498.235,A -85,B 0,C 180,E1 -10704.612,E2 -10704.612} C_VEL
LIN {X 0,Y 411.302,Z 501.105,A -85,B 0,C 180,E1 -10706.081,E2 -10706.081} C_VEL
LIN {X 0,Y 411.335,Z 502.457,A -85,B 0,C 180,E1 -10707.062,E2 -10707.062} C_VEL
LIN {X 0,Y 411.181,Z 503.441,A -85,B 0,C 180,E1 -10708.041,E2 -10708.041} C_VEL
LIN {X 0,Y 411.235,Z 504.22,A -85,B 0,C 180,E1 -10709.857,E2 -10709.857} C_VEL
LIN {X 0,Y 410.578,Z 504.354,A -85,B 0,C 180,E1 -10710.677,E2 -10710.677} C_VEL
LIN {X 0,Y 407.706,Z 504.163,A -85,B 0,C 180,E1 -10712.008,E2 -10712.008} C_VEL
LIN {X 0,Y 404.878,Z 503.122,A -85,B 0,C 180,E1 -10713.346,E2 -10713.346} C_VEL
LIN {X 0,Y 404.302,Z 501.922,A -85,B 0,C 180,E1 -10714.163,E2 -10714.163} C_VEL
LIN {X 0,Y 404.661,Z 498.259,A -85,B 0,C 180,E1 -10715.981,E2 -10715.981} C_VEL
LIN {X 0,Y 405.205,Z 494.072,A -85,B 0,C 180,E1 -10717.474,E2 -10717.474} C_VEL
LIN {X 0,Y 405.561,Z 488.764,A -85,B 0,C 180,E1 -10718.972,E2 -10718.972} C_VEL
LIN {X 0,Y 406.247,Z 482.085,A -85,B 0,C 180,E1 -10720.466,E2 -10720.466} C_VEL
LIN {X 0,Y 406.94,Z 473.742,A -85,B 0,C 180,E1 -10721.961,E2 -10721.961} C_VEL
LIN {X 0,Y 407.534,Z 465.161,A -85,B 0,C 180,E1 -10723.208,E2 -10723.208} C_VEL
LIN {X 0,Y 408.268,Z 456.847,A -85,B 0,C 180,E1 -10724.199,E2 -10724.199} C_VEL
LIN {X 0,Y 408.966,Z 446.492,A -85,B 0,C 180,E1 -10725.215,E2 -10725.215} C_VEL
LIN {X 0,Y 409.529,Z 434.581,A -85,B 0,C 180,E1 -10726.144,E2 -10726.144} C_VEL
LIN {X 0,Y 409.937,Z 422.029,A -85,B 0,C 180,E1 -10726.874,E2 -10726.874} C_VEL
LIN {X 0,Y 410.161,Z 408.847,A -85,B 0,C 180,E1 -10727.417,E2 -10727.417} C_VEL
LIN {X 0,Y 410.182,Z 396.176,A -85,B 0,C 180,E1 -10727.737,E2 -10727.737} C_VEL
LIN {X 0,Y 410.706,Z 338.067,A -85,B 0,C 180,E1 -10728.767,E2 -10728.767} C_VEL
LIN {X 0,Y 404.464,Z 322.324,A -85,B 0,C 180,E1 -10729.391,E2 -10729.391} C_VEL
LIN {X 0,Y 404.224,Z 321.28,A -85,B 0,C 180,E1 -10729.568,E2 -10729.568} C_VEL
LIN {X 0,Y 404.146,Z 321.124,A -85,B 0,C 180,E1 -10732.83,E2 -10732.83} C_VEL
LIN {X 0,Y 404.13,Z 321.133,A -85,B 0,C 180,E1 -10735.77,E2 -10735.77} C_VEL
LIN {X 0,Y 404.152,Z 321.138,A -85,B 0,C 180,E1 -10739.602,E2 -10739.602} C_VEL
LIN {X 0,Y 404.165,Z 321.137,A -85,B 0,C 180,E1 -10743.418,E2 -10743.418} C_VEL
LIN {X 0,Y 404.132,Z 321.14,A -85,B 0,C 180,E1 -10746.247,E2 -10746.247} C_VEL
LIN {X 0,Y 404.131,Z 321.139,A -85,B 0,C 180,E1 -10748.759,E2 -10748.759} C_VEL
LIN {X 0,Y 404.102,Z 321.141,A -85,B 0,C 180,E1 -10751.596,E2 -10751.596} C_VEL
LIN {X 0,Y 404.14,Z 321.131,A -85,B 0,C 180,E1 -10754.521,E2 -10754.521} C_VEL
LIN {X 0,Y 404.116,Z 321.145,A -85,B 0,C 180,E1 -10757.293,E2 -10757.293} C_VEL
LIN {X 0,Y 404.129,Z 321.127,A -85,B 0,C 180,E1 -10759.95,E2 -10759.95} C_VEL
LIN {X 0,Y 404.129,Z 321.14,A -85,B 0,C 180,E1 -10763.125,E2 -10763.125} C_VEL
LIN {X 0,Y 404.133,Z 321.144,A -85,B 0,C 180,E1 -10766.186,E2 -10766.186} C_VEL
LIN {X 0,Y 404.136,Z 321.113,A -85,B 0,C 180,E1 -10769.714,E2 -10769.714} C_VEL
LIN {X 0,Y 404.098,Z 321.139,A -85,B 0,C 180,E1 -10773.116,E2 -10773.116} C_VEL
LIN {X 0,Y 404.141,Z 321.147,A -85,B 0,C 180,E1 -10776.424,E2 -10776.424} C_VEL
LIN {X 0,Y 404.149,Z 321.132,A -85,B 0,C 180,E1 -10779.888,E2 -10779.888} C_VEL
LIN {X 0,Y 404.209,Z 321.131,A -85,B 0,C 180,E1 -10782.993,E2 -10782.993} C_VEL
LIN {X 0,Y 404.277,Z 321.123,A -85,B 0,C 180,E1 -10786.939,E2 -10786.939} C_VEL
LIN {X 0,Y 404.24,Z 321.13,A -85,B 0,C 180,E1 -10789.988,E2 -10789.988} C_VEL
LIN {X 0,Y 404.329,Z 321.112,A -85,B 0,C 180,E1 -10793.011,E2 -10793.011} C_VEL
LIN {X 0,Y 404.25,Z 321.128,A -85,B 0,C 180,E1 -10795.013,E2 -10795.013} C_VEL
LIN {X 0,Y 404.466,Z 321.098,A -85,B 0,C 180,E1 -10798.008,E2 -10798.008} C_VEL
LIN {X 0,Y 404.462,Z 321.101,A -85,B 0,C 180,E1 -10801.992,E2 -10801.992} C_VEL
LIN {X 0,Y 404.386,Z 321.102,A -85,B 0,C 180,E1 -10805.985,E2 -10805.985} C_VEL
LIN {X 0,Y 404.253,Z 321.126,A -85,B 0,C 180,E1 -10809.002,E2 -10809.002} C_VEL
LIN {X 0,Y 404.241,Z 321.124,A -85,B 0,C 180,E1 -10812.042,E2 -10812.042} C_VEL
LIN {X 0,Y 404.198,Z 321.133,A -85,B 0,C 180,E1 -10815.118,E2 -10815.118} C_VEL
LIN {X 0,Y 404.196,Z 321.129,A -85,B 0,C 180,E1 -10818.239,E2 -10818.239} C_VEL
LIN {X 0,Y 404.131,Z 321.124,A -85,B 0,C 180,E1 -10821.42,E2 -10821.42} C_VEL
LIN {X 0,Y 404.142,Z 321.142,A -85,B 0,C 180,E1 -10824.668,E2 -10824.668} C_VEL
LIN {X 0,Y 404.116,Z 321.133,A -85,B 0,C 180,E1 -10828.006,E2 -10828.006} C_VEL
LIN {X 0,Y 404.139,Z 321.141,A -85,B 0,C 180,E1 -10830.286,E2 -10830.286} C_VEL
LIN {X 0,Y 404.132,Z 321.138,A -85,B 0,C 180,E1 -10833.814,E2 -10833.814} C_VEL
LIN {X 0,Y 404.126,Z 321.144,A -85,B 0,C 180,E1 -10836.874,E2 -10836.874} C_VEL
LIN {X 0,Y 404.112,Z 321.141,A -85,B 0,C 180,E1 -10840.075,E2 -10840.075} C_VEL
LIN {X 0,Y 404.138,Z 321.136,A -85,B 0,C 180,E1 -10843.083,E2 -10843.083} C_VEL
LIN {X 0,Y 404.115,Z 321.125,A -85,B 0,C 180,E1 -10845.923,E2 -10845.923} C_VEL
LIN {X 0,Y 404.098,Z 321.145,A -85,B 0,C 180,E1 -10848.633,E2 -10848.633} C_VEL
LIN {X 0,Y 404.134,Z 321.137,A -85,B 0,C 180,E1 -10851.496,E2 -10851.496} C_VEL
LIN {X 0,Y 404.17,Z 321.132,A -85,B 0,C 180,E1 -10854.983,E2 -10854.983} C_VEL
LIN {X 0,Y 404.195,Z 321.386,A -85,B 0,C 180,E1 -10857.218,E2 -10857.218} C_VEL
LIN {X 0,Y 407.752,Z 336.594,A -85,B 0,C 180,E1 -10860.011,E2 -10860.011} C_VEL
LIN {X 0,Y 409.119,Z 343.692,A -85,B 0,C 180,E1 -10861.25,E2 -10861.25} C_VEL
LIN {X 0,Y 408.007,Z 361.098,A -85,B 0,C 180,E1 -10863.989,E2 -10863.989} C_VEL
LIN {X 0,Y 406.505,Z 382.846,A -85,B 0,C 180,E1 -10867.377,E2 -10867.377} C_VEL
LIN {X 0,Y 405.475,Z 401.109,A -85,B 0,C 180,E1 -10870.197,E2 -10870.197} C_VEL
LIN {X 0,Y 409.045,Z 432.986,A -85,B 0,C 180,E1 -10870.964,E2 -10870.964} C_VEL
LIN {X 0,Y 409.782,Z 443.254,A -85,B 0,C 180,E1 -10871.183,E2 -10871.183} C_VEL
LIN {X 0,Y 408.904,Z 511.608,A -85,B 0,C 180,E1 -10872.399,E2 -10872.399} C_VEL
LIN {X 0,Y 408.412,Z 524.914,A -85,B 0,C 180,E1 -10872.829,E2 -10872.829} C_VEL
LIN {X 0,Y 407.535,Z 538.249,A -85,B 0,C 180,E1 -10873.469,E2 -10873.469} C_VEL
LIN {X 0,Y 406.726,Z 549.484,A -85,B 0,C 180,E1 -10874.208,E2 -10874.208} C_VEL
LIN {X 0,Y 405.684,Z 561.181,A -85,B 0,C 180,E1 -10875.195,E2 -10875.195} C_VEL
LIN {X 0,Y 404.906,Z 572.529,A -85,B 0,C 180,E1 -10876.41,E2 -10876.41} C_VEL
LIN {X 0,Y 404.439,Z 580.48,A -85,B 0,C 180,E1 -10877.455,E2 -10877.455} C_VEL
LIN {X 0,Y 403.853,Z 588.514,A -85,B 0,C 180,E1 -10878.71,E2 -10878.71} C_VEL
LIN {X 0,Y 403.465,Z 596.405,A -85,B 0,C 180,E1 -10880.222,E2 -10880.222} C_VEL
LIN {X 0,Y 403.345,Z 603.722,A -85,B 0,C 180,E1 -10881.987,E2 -10881.987} C_VEL
LIN {X 0,Y 403.345,Z 608.054,A -85,B 0,C 180,E1 -10883.308,E2 -10883.308} C_VEL
LIN {X 0,Y 403.493,Z 612.367,A -85,B 0,C 180,E1 -10885.004,E2 -10885.004} C_VEL
LIN {X 0,Y 403.626,Z 614.314,A -85,B 0,C 180,E1 -10886.006,E2 -10886.006} C_VEL
LIN {X 0,Y 403.596,Z 615.757,A -85,B 0,C 180,E1 -10887.006,E2 -10887.006} C_VEL
LIN {X 0,Y 403.888,Z 617.459,A -85,B 0,C 180,E1 -10889.003,E2 -10889.003} C_VEL
LIN {X 0,Y 403.91,Z 617.686,A -85,B 0,C 180,E1 -10890,E2 -10890} C_VEL
LIN {X 0,Y 403.888,Z 617.458,A -85,B 0,C 180,E1 -10890.997,E2 -10890.997} C_VEL
LIN {X 0,Y 403.596,Z 615.755,A -85,B 0,C 180,E1 -10892.994,E2 -10892.994} C_VEL
LIN {X 0,Y 403.626,Z 614.31,A -85,B 0,C 180,E1 -10893.994,E2 -10893.994} C_VEL
LIN {X 0,Y 403.41,Z 611.237,A -85,B 0,C 180,E1 -10895.498,E2 -10895.498} C_VEL
LIN {X 0,Y 403.355,Z 607.112,A -85,B 0,C 180,E1 -10897.005,E2 -10897.005} C_VEL
LIN {X 0,Y 403.362,Z 600.786,A -85,B 0,C 180,E1 -10898.769,E2 -10898.769} C_VEL
LIN {X 0,Y 403.551,Z 593.912,A -85,B 0,C 180,E1 -10900.283,E2 -10900.283} C_VEL
LIN {X 0,Y 404.01,Z 585.432,A -85,B 0,C 180,E1 -10901.794,E2 -10901.794} C_VEL
LIN {X 0,Y 404.678,Z 576.781,A -85,B 0,C 180,E1 -10903.048,E2 -10903.048} C_VEL
LIN {X 0,Y 405.361,Z 566.105,A -85,B 0,C 180,E1 -10904.303,E2 -10904.303} C_VEL
LIN {X 0,Y 406.188,Z 555.599,A -85,B 0,C 180,E1 -10905.299,E2 -10905.299} C_VEL
LIN {X 0,Y 407.087,Z 544.115,A -85,B 0,C 180,E1 -10906.163,E2 -10906.163} C_VEL
LIN {X 0,Y 407.92,Z 532.345,A -85,B 0,C 180,E1 -10906.837,E2 -10906.837} C_VEL
LIN {X 0,Y 408.684,Z 518.818,A -85,B 0,C 180,E1 -10907.385,E2 -10907.385} C_VEL
LIN {X 0,Y 409.03,Z 505.396,A -85,B 0,C 180,E1 -10907.724,E2 -10907.724} C_VEL
LIN {X 0,Y 409.754,Z 440.666,A -85,B 0,C 180,E1 -10908.858,E2 -10908.858} C_VEL
LIN {X 0,Y 405.542,Z 401.766,A -85,B 0,C 180,E1 -10909.767,E2 -10909.767} C_VEL
LIN {X 0,Y 405.495,Z 400.315,A -85,B 0,C 180,E1 -10909.885,E2 -10909.885} C_VEL
LIN {X 0,Y 406.962,Z 375.504,A -85,B 0,C 180,E1 -10913.754,E2 -10913.754} C_VEL
LIN {X 0,Y 408.447,Z 353.906,A -85,B 0,C 180,E1 -10917.127,E2 -10917.127} C_VEL
LIN {X 0,Y 409.118,Z 343.625,A -85,B 0,C 180,E1 -10918.75,E2 -10918.75} C_VEL
LIN {X 0,Y 406.487,Z 330.931,A -85,B 0,C 180,E1 -10920.992,E2 -10920.992} C_VEL
LIN {X 0,Y 404.176,Z 321.26,A -85,B 0,C 180,E1 -10922.817,E2 -10922.817} C_VEL
LIN {X 0,Y 404.131,Z 321.137,A -85,B 0,C 180,E1 -10926.247,E2 -10926.247} C_VEL
LIN {X 0,Y 404.129,Z 321.135,A -85,B 0,C 180,E1 -10928.759,E2 -10928.759} C_VEL
LIN {X 0,Y 404.102,Z 321.148,A -85,B 0,C 180,E1 -10931.596,E2 -10931.596} C_VEL
LIN {X 0,Y 404.139,Z 321.118,A -85,B 0,C 180,E1 -10934.521,E2 -10934.521} C_VEL
LIN {X 0,Y 404.118,Z 321.141,A -85,B 0,C 180,E1 -10937.293,E2 -10937.293} C_VEL
LIN {X 0,Y 404.128,Z 321.137,A -85,B 0,C 180,E1 -10939.95,E2 -10939.95} C_VEL
LIN {X 0,Y 404.125,Z 321.099,A -85,B 0,C 180,E1 -10943.126,E2 -10943.126} C_VEL
LIN {X 0,Y 404.132,Z 321.137,A -85,B 0,C 180,E1 -10946.186,E2 -10946.186} C_VEL
LIN {X 0,Y 404.139,Z 321.14,A -85,B 0,C 180,E1 -10949.714,E2 -10949.714} C_VEL
LIN {X 0,Y 404.123,Z 321.137,A -85,B 0,C 180,E1 -10953.118,E2 -10953.118} C_VEL
LIN {X 0,Y 404.143,Z 321.138,A -85,B 0,C 180,E1 -10956.424,E2 -10956.424} C_VEL
LIN {X 0,Y 404.185,Z 321.118,A -85,B 0,C 180,E1 -10959.874,E2 -10959.874} C_VEL
LIN {X 0,Y 404.21,Z 321.131,A -85,B 0,C 180,E1 -10962.993,E2 -10962.993} C_VEL
LIN {X 0,Y 404.276,Z 321.113,A -85,B 0,C 180,E1 -10966.939,E2 -10966.939} C_VEL
LIN {X 0,Y 404.246,Z 321.132,A -85,B 0,C 180,E1 -10969.988,E2 -10969.988} C_VEL
LIN {X 0,Y 404.374,Z 321.106,A -85,B 0,C 180,E1 -10973.012,E2 -10973.012} C_VEL
LIN {X 0,Y 404.258,Z 321.119,A -85,B 0,C 180,E1 -10975.013,E2 -10975.013} C_VEL
LIN {X 0,Y 404.462,Z 321.102,A -85,B 0,C 180,E1 -10978.008,E2 -10978.008} C_VEL
LIN {X 0,Y 404.339,Z 321.103,A -85,B 0,C 180,E1 -10980.996,E2 -10980.996} C_VEL
LIN {X 0,Y 404.391,Z 321.107,A -85,B 0,C 180,E1 -10982.989,E2 -10982.989} C_VEL
LIN {X 0,Y 404.333,Z 321.111,A -85,B 0,C 180,E1 -10986.989,E2 -10986.989} C_VEL
LIN {X 0,Y 404.248,Z 321.129,A -85,B 0,C 180,E1 -10990.012,E2 -10990.012} C_VEL
LIN {X 0,Y 404.26,Z 321.125,A -85,B 0,C 180,E1 -10993.212,E2 -10993.212} C_VEL
LIN {X 0,Y 404.21,Z 321.131,A -85,B 0,C 180,E1 -10997.007,E2 -10997.007} C_VEL
LIN {X 0,Y 404.158,Z 321.13,A -85,B 0,C 180,E1 -11000.352,E2 -11000.352} C_VEL
LIN {X 0,Y 404.143,Z 321.146,A -85,B 0,C 180,E1 -11003.576,E2 -11003.576} C_VEL
LIN {X 0,Y 404.098,Z 321.139,A -85,B 0,C 180,E1 -11006.884,E2 -11006.884} C_VEL
LIN {X 0,Y 404.136,Z 321.112,A -85,B 0,C 180,E1 -11010.286,E2 -11010.286} C_VEL
LIN {X 0,Y 404.133,Z 321.145,A -85,B 0,C 180,E1 -11013.814,E2 -11013.814} C_VEL
LIN {X 0,Y 404.129,Z 321.139,A -85,B 0,C 180,E1 -11016.875,E2 -11016.875} C_VEL
LIN {X 0,Y 404.113,Z 321.127,A -85,B 0,C 180,E1 -11020.075,E2 -11020.075} C_VEL
LIN {X 0,Y 404.138,Z 321.144,A -85,B 0,C 180,E1 -11023.083,E2 -11023.083} C_VEL
LIN {X 0,Y 404.117,Z 321.13,A -85,B 0,C 180,E1 -11025.923,E2 -11025.923} C_VEL
LIN {X 0,Y 404.098,Z 321.142,A -85,B 0,C 180,E1 -11028.633,E2 -11028.633} C_VEL
LIN {X 0,Y 404.136,Z 321.136,A -85,B 0,C 180,E1 -11031.496,E2 -11031.496} C_VEL
LIN {X 0,Y 404.172,Z 321.139,A -85,B 0,C 180,E1 -11034.983,E2 -11034.983} C_VEL
LIN {X 0,Y 404.133,Z 321.14,A -85,B 0,C 180,E1 -11038.444,E2 -11038.444} C_VEL
LIN {X 0,Y 404.147,Z 321.132,A -85,B 0,C 180,E1 -11040.863,E2 -11040.863} C_VEL
LIN {X 0,Y 404.151,Z 321.14,A -85,B 0,C 180,E1 -11044.724,E2 -11044.724} C_VEL
LIN {X 0,Y 404.166,Z 321.122,A -85,B 0,C 180,E1 -11047.508,E2 -11047.508} C_VEL
LIN {X 0,Y 404.269,Z 321.306,A -85,B 0,C 180,E1 -11050.545,E2 -11050.545} C_VEL
LIN {X 0,Y 404.485,Z 322.31,A -85,B 0,C 180,E1 -11050.71,E2 -11050.71} C_VEL
LIN {X 0,Y 410.721,Z 338.059,A -85,B 0,C 180,E1 -11051.333,E2 -11051.333} C_VEL
LIN {X 0,Y 410.238,Z 402.144,A -85,B 0,C 180,E1 -11052.49,E2 -11052.49} C_VEL
LIN {X 0,Y 410.077,Z 414.82,A -85,B 0,C 180,E1 -11052.901,E2 -11052.901} C_VEL
LIN {X 0,Y 409.764,Z 427.171,A -85,B 0,C 180,E1 -11053.498,E2 -11053.498} C_VEL
LIN {X 0,Y 409.342,Z 438.417,A -85,B 0,C 180,E1 -11054.228,E2 -11054.228} C_VEL
LIN {X 0,Y 408.612,Z 449.825,A -85,B 0,C 180,E1 -11055.177,E2 -11055.177} C_VEL
LIN {X 0,Y 407.854,Z 460.387,A -85,B 0,C 180,E1 -11056.295,E2 -11056.295} C_VEL
LIN {X 0,Y 407.212,Z 469.857,A -85,B 0,C 180,E1 -11057.542,E2 -11057.542} C_VEL
LIN {X 0,Y 406.549,Z 477.614,A -85,B 0,C 180,E1 -11058.786,E2 -11058.786} C_VEL
LIN {X 0,Y 405.904,Z 485.291,A -85,B 0,C 180,E1 -11060.306,E2 -11060.306} C_VEL
LIN {X 0,Y 405.409,Z 491.046,A -85,B 0,C 180,E1 -11061.726,E2 -11061.726} C_VEL
LIN {X 0,Y 405.11,Z 495.318,A -85,B 0,C 180,E1 -11063.025,E2 -11063.025} C_VEL
LIN {X 0,Y 404.615,Z 499.214,A -85,B 0,C 180,E1 -11064.518,E2 -11064.518} C_VEL
LIN {X 0,Y 404.286,Z 502.085,A -85,B 0,C 180,E1 -11066.013,E2 -11066.013} C_VEL
LIN {X 0,Y 404.316,Z 503.435,A -85,B 0,C 180,E1 -11067.011,E2 -11067.011} C_VEL
LIN {X 0,Y 404.159,Z 504.419,A -85,B 0,C 180,E1 -11068.007,E2 -11068.007} C_VEL
LIN {X 0,Y 404.211,Z 505.198,A -85,B 0,C 180,E1 -11069.857,E2 -11069.857} C_VEL
LIN {X 0,Y 404.233,Z 505.047,A -85,B 0,C 180,E1 -11070.996,E2 -11070.996} C_VEL
LIN {X 0,Y 404.158,Z 504.493,A -85,B 0,C 180,E1 -11071.993,E2 -11071.993} C_VEL
LIN {X 0,Y 404.313,Z 503.539,A -85,B 0,C 180,E1 -11072.989,E2 -11072.989} C_VEL
LIN {X 0,Y 404.302,Z 501.922,A -85,B 0,C 180,E1 -11074.163,E2 -11074.163} C_VEL
LIN {X 0,Y 403.801,Z 500.59,A -85,B 0,C 180,E1 -11074.974,E2 -11074.974} C_VEL
LIN {X 0,Y 401.322,Z 498.104,A -85,B 0,C 180,E1 -11076.295,E2 -11076.295} C_VEL
LIN {X 0,Y 399.238,Z 495.66,A -85,B 0,C 180,E1 -11077.34,E2 -11077.34} C_VEL
LIN {X 0,Y 398.421,Z 493.393,A -85,B 0,C 180,E1 -11078.12,E2 -11078.12} C_VEL
LIN {X 0,Y 398.398,Z 492.521,A -85,B 0,C 180,E1 -11078.376,E2 -11078.376} C_VEL
LIN {X 0,Y 398.937,Z 486.586,A -85,B 0,C 180,E1 -11079.89,E2 -11079.89} C_VEL
LIN {X 0,Y 399.73,Z 479.134,A -85,B 0,C 180,E1 -11081.408,E2 -11081.408} C_VEL
LIN {X 0,Y 400.332,Z 471.508,A -85,B 0,C 180,E1 -11082.676,E2 -11082.676} C_VEL
LIN {X 0,Y 401.037,Z 461.132,A -85,B 0,C 180,E1 -11084.072,E2 -11084.072} C_VEL
LIN {X 0,Y 401.91,Z 450.502,A -85,B 0,C 180,E1 -11085.206,E2 -11085.206} C_VEL
LIN {X 0,Y 402.577,Z 439.67,A -85,B 0,C 180,E1 -11086.123,E2 -11086.123} C_VEL
LIN {X 0,Y 403.16,Z 426.952,A -85,B 0,C 180,E1 -11086.951,E2 -11086.951} C_VEL
LIN {X 0,Y 403.463,Z 414.315,A -85,B 0,C 180,E1 -11087.552,E2 -11087.552} C_VEL
LIN {X 0,Y 403.546,Z 401.742,A -85,B 0,C 180,E1 -11087.941,E2 -11087.941} C_VEL
LIN {X 0,Y 404.016,Z 339.665,A -85,B 0,C 180,E1 -11089.077,E2 -11089.077} C_VEL
LIN {X 0,Y 397.345,Z 323.001,A -85,B 0,C 180,E1 -11089.767,E2 -11089.767} C_VEL
LIN {X 0,Y 397.142,Z 322.087,A -85,B 0,C 180,E1 -11089.981,E2 -11089.981} C_VEL
LIN {X 0,Y 397.095,Z 322.003,A -85,B 0,C 180,E1 -11093.026,E2 -11093.026} C_VEL
LIN {X 0,Y 397.07,Z 322.001,A -85,B 0,C 180,E1 -11096.262,E2 -11096.262} C_VEL
LIN {X 0,Y 397.096,Z 322.017,A -85,B 0,C 180,E1 -11099.862,E2 -11099.862} C_VEL
LIN {X 0,Y 397.108,Z 322.014,A -85,B 0,C 180,E1 -11103.273,E2 -11103.273} C_VEL
LIN {X 0,Y 397.092,Z 322.008,A -85,B 0,C 180,E1 -11106.995,E2 -11106.995} C_VEL
LIN {X 0,Y 397.052,Z 322.028,A -85,B 0,C 180,E1 -11110.437,E2 -11110.437} C_VEL
LIN {X 0,Y 397.083,Z 322.004,A -85,B 0,C 180,E1 -11113.65,E2 -11113.65} C_VEL
LIN {X 0,Y 397.087,Z 322.024,A -85,B 0,C 180,E1 -11116.522,E2 -11116.522} C_VEL
LIN {X 0,Y 397.082,Z 321.998,A -85,B 0,C 180,E1 -11120.419,E2 -11120.419} C_VEL
LIN {X 0,Y 397.091,Z 322.013,A -85,B 0,C 180,E1 -11123.004,E2 -11123.004} C_VEL
LIN {X 0,Y 397.093,Z 322.022,A -85,B 0,C 180,E1 -11126.286,E2 -11126.286} C_VEL
LIN {X 0,Y 397.07,Z 321.996,A -85,B 0,C 180,E1 -11129.117,E2 -11129.117} C_VEL
LIN {X 0,Y 397.055,Z 322.001,A -85,B 0,C 180,E1 -11132.251,E2 -11132.251} C_VEL
LIN {X 0,Y 397.096,Z 322.021,A -85,B 0,C 180,E1 -11134.864,E2 -11134.864} C_VEL
LIN {X 0,Y 397.086,Z 322.017,A -85,B 0,C 180,E1 -11138.181,E2 -11138.181} C_VEL
LIN {X 0,Y 397.148,Z 322.011,A -85,B 0,C 180,E1 -11141.426,E2 -11141.426} C_VEL
LIN {X 0,Y 397.161,Z 322.002,A -85,B 0,C 180,E1 -11144.607,E2 -11144.607} C_VEL
LIN {X 0,Y 397.211,Z 322.002,A -85,B 0,C 180,E1 -11147.742,E2 -11147.742} C_VEL
LIN {X 0,Y 397.221,Z 321.996,A -85,B 0,C 180,E1 -11150.837,E2 -11150.837} C_VEL
LIN {X 0,Y 397.308,Z 321.988,A -85,B 0,C 180,E1 -11153.907,E2 -11153.907} C_VEL
LIN {X 0,Y 397.435,Z 321.974,A -85,B 0,C 180,E1 -11157.973,E2 -11157.973} C_VEL
LIN {X 0,Y 397.431,Z 321.977,A -85,B 0,C 180,E1 -11162.027,E2 -11162.027} C_VEL
LIN {X 0,Y 397.34,Z 321.979,A -85,B 0,C 180,E1 -11166.092,E2 -11166.092} C_VEL
LIN {X 0,Y 397.223,Z 322.002,A -85,B 0,C 180,E1 -11169.163,E2 -11169.163} C_VEL
LIN {X 0,Y 397.207,Z 321.997,A -85,B 0,C 180,E1 -11172.259,E2 -11172.259} C_VEL
LIN {X 0,Y 397.171,Z 322.008,A -85,B 0,C 180,E1 -11175.392,E2 -11175.392} C_VEL
LIN {X 0,Y 397.15,Z 322.003,A -85,B 0,C 180,E1 -11178.574,E2 -11178.574} C_VEL
LIN {X 0,Y 397.088,Z 322.004,A -85,B 0,C 180,E1 -11181.819,E2 -11181.819} C_VEL
LIN {X 0,Y 397.091,Z 322.019,A -85,B 0,C 180,E1 -11185.136,E2 -11185.136} C_VEL
LIN {X 0,Y 397.067,Z 322.01,A -85,B 0,C 180,E1 -11188.548,E2 -11188.548} C_VEL
LIN {X 0,Y 397.076,Z 322.025,A -85,B 0,C 180,E1 -11191.837,E2 -11191.837} C_VEL
LIN {X 0,Y 397.111,Z 322.008,A -85,B 0,C 180,E1 -11194.495,E2 -11194.495} C_VEL
LIN {X 0,Y 397.084,Z 322.018,A -85,B 0,C 180,E1 -11198.277,E2 -11198.277} C_VEL
LIN {X 0,Y 397.048,Z 322.028,A -85,B 0,C 180,E1 -11201.977,E2 -11201.977} C_VEL
LIN {X 0,Y 397.08,Z 321.994,A -85,B 0,C 180,E1 -11205.07,E2 -11205.07} C_VEL
LIN {X 0,Y 397.047,Z 322.03,A -85,B 0,C 180,E1 -11208.024,E2 -11208.024} C_VEL
LIN {X 0,Y 397.086,Z 322.017,A -85,B 0,C 180,E1 -11211.724,E2 -11211.724} C_VEL
LIN {X 0,Y 397.114,Z 322.018,A -85,B 0,C 180,E1 -11215.506,E2 -11215.506} C_VEL
LIN {X 0,Y 397.157,Z 322.207,A -85,B 0,C 180,E1 -11216.864,E2 -11216.864} C_VEL
LIN {X 0,Y 400.798,Z 337.87,A -85,B 0,C 180,E1 -11219.807,E2 -11219.807} C_VEL
LIN {X 0,Y 402.26,Z 345.175,A -85,B 0,C 180,E1 -11221.111,E2 -11221.111} C_VEL
LIN {X 0,Y 400.948,Z 363.285,A -85,B 0,C 180,E1 -11224.011,E2 -11224.011} C_VEL
LIN {X 0,Y 399.514,Z 383.541,A -85,B 0,C 180,E1 -11227.232,E2 -11227.232} C_VEL
LIN {X 0,Y 398.526,Z 400.1,A -85,B 0,C 180,E1 -11229.836,E2 -11229.836} C_VEL
LIN {X 0,Y 402.329,Z 433.977,A -85,B 0,C 180,E1 -11230.669,E2 -11230.669} C_VEL
LIN {X 0,Y 403.037,Z 443.668,A -85,B 0,C 180,E1 -11230.881,E2 -11230.881} C_VEL
LIN {X 0,Y 402.125,Z 510.63,A -85,B 0,C 180,E1 -11232.092,E2 -11232.092} C_VEL
LIN {X 0,Y 401.607,Z 523.93,A -85,B 0,C 180,E1 -11232.529,E2 -11232.529} C_VEL
LIN {X 0,Y 400.715,Z 537.264,A -85,B 0,C 180,E1 -11233.179,E2 -11233.179} C_VEL
LIN {X 0,Y 399.874,Z 548.497,A -85,B 0,C 180,E1 -11233.93,E2 -11233.93} C_VEL
LIN {X 0,Y 398.77,Z 560.189,A -85,B 0,C 180,E1 -11234.933,E2 -11234.933} C_VEL
LIN {X 0,Y 397.956,Z 571.47,A -85,B 0,C 180,E1 -11236.159,E2 -11236.159} C_VEL
LIN {X 0,Y 397.283,Z 581.195,A -85,B 0,C 180,E1 -11237.485,E2 -11237.485} C_VEL
LIN {X 0,Y 396.742,Z 588.933,A -85,B 0,C 180,E1 -11238.764,E2 -11238.764} C_VEL
LIN {X 0,Y 396.364,Z 596.561,A -85,B 0,C 180,E1 -11240.303,E2 -11240.303} C_VEL
LIN {X 0,Y 396.276,Z 602.73,A -85,B 0,C 180,E1 -11241.843,E2 -11241.843} C_VEL
LIN {X 0,Y 396.287,Z 607.349,A -85,B 0,C 180,E1 -11243.286,E2 -11243.286} C_VEL
LIN {X 0,Y 396.405,Z 611.378,A -85,B 0,C 180,E1 -11244.914,E2 -11244.914} C_VEL
LIN {X 0,Y 396.563,Z 613.329,A -85,B 0,C 180,E1 -11245.935,E2 -11245.935} C_VEL
LIN {X 0,Y 396.55,Z 614.776,A -85,B 0,C 180,E1 -11246.952,E2 -11246.952} C_VEL
LIN {X 0,Y 396.857,Z 616.481,A -85,B 0,C 180,E1 -11248.985,E2 -11248.985} C_VEL
LIN {X 0,Y 396.885,Z 616.708,A -85,B 0,C 180,E1 -11250,E2 -11250} C_VEL
LIN {X 0,Y 396.857,Z 616.479,A -85,B 0,C 180,E1 -11251.015,E2 -11251.015} C_VEL
LIN {X 0,Y 396.551,Z 614.773,A -85,B 0,C 180,E1 -11253.048,E2 -11253.048} C_VEL
LIN {X 0,Y 396.564,Z 613.324,A -85,B 0,C 180,E1 -11254.065,E2 -11254.065} C_VEL
LIN {X 0,Y 396.343,Z 610.248,A -85,B 0,C 180,E1 -11255.597,E2 -11255.597} C_VEL
LIN {X 0,Y 396.288,Z 606.12,A -85,B 0,C 180,E1 -11257.131,E2 -11257.131} C_VEL
LIN {X 0,Y 396.29,Z 599.789,A -85,B 0,C 180,E1 -11258.927,E2 -11258.927} C_VEL
LIN {X 0,Y 396.521,Z 592.916,A -85,B 0,C 180,E1 -11260.467,E2 -11260.467} C_VEL
LIN {X 0,Y 396.962,Z 584.427,A -85,B 0,C 180,E1 -11262.007,E2 -11262.007} C_VEL
LIN {X 0,Y 397.646,Z 575.773,A -85,B 0,C 180,E1 -11263.283,E2 -11263.283} C_VEL
LIN {X 0,Y 398.407,Z 565.103,A -85,B 0,C 180,E1 -11264.559,E2 -11264.559} C_VEL
LIN {X 0,Y 399.275,Z 554.597,A -85,B 0,C 180,E1 -11265.571,E2 -11265.571} C_VEL
LIN {X 0,Y 400.251,Z 543.119,A -85,B 0,C 180,E1 -11266.447,E2 -11266.447} C_VEL
LIN {X 0,Y 401.095,Z 531.345,A -85,B 0,C 180,E1 -11267.133,E2 -11267.133} C_VEL
LIN {X 0,Y 401.853,Z 518.735,A -85,B 0,C 180,E1 -11267.657,E2 -11267.657} C_VEL
LIN {X 0,Y 402.225,Z 505.932,A -85,B 0,C 180,E1 -11268.002,E2 -11268.002} C_VEL
LIN {X 0,Y 403.006,Z 441.161,A -85,B 0,C 180,E1 -11269.158,E2 -11269.158} C_VEL
LIN {X 0,Y 398.949,Z 403.664,A -85,B 0,C 180,E1 -11270.047,E2 -11270.047} C_VEL
LIN {X 0,Y 398.538,Z 399.807,A -85,B 0,C 180,E1 -11270.18,E2 -11270.18} C_VEL
LIN {X 0,Y 400.02,Z 375.768,A -85,B 0,C 180,E1 -11273.993,E2 -11273.993} C_VEL
LIN {X 0,Y 401.566,Z 354.693,A -85,B 0,C 180,E1 -11277.349,E2 -11277.349} C_VEL
LIN {X 0,Y 402.228,Z 345.118,A -85,B 0,C 180,E1 -11278.888,E2 -11278.888} C_VEL
LIN {X 0,Y 399.885,Z 333.725,A -85,B 0,C 180,E1 -11280.934,E2 -11280.934} C_VEL
LIN {X 0,Y 397.14,Z 322.13,A -85,B 0,C 180,E1 -11283.156,E2 -11283.156} C_VEL
LIN {X 0,Y 397.09,Z 322.011,A -85,B 0,C 180,E1 -11285.736,E2 -11285.736} C_VEL
LIN {X 0,Y 397.088,Z 322.01,A -85,B 0,C 180,E1 -11288.854,E2 -11288.854} C_VEL
LIN {X 0,Y 397.051,Z 322.028,A -85,B 0,C 180,E1 -11292.269,E2 -11292.269} C_VEL
LIN {X 0,Y 397.08,Z 321.994,A -85,B 0,C 180,E1 -11295.069,E2 -11295.069} C_VEL
LIN {X 0,Y 397.048,Z 322.03,A -85,B 0,C 180,E1 -11298.023,E2 -11298.023} C_VEL
LIN {X 0,Y 397.084,Z 321.986,A -85,B 0,C 180,E1 -11301.723,E2 -11301.723} C_VEL
LIN {X 0,Y 397.111,Z 322.001,A -85,B 0,C 180,E1 -11305.505,E2 -11305.505} C_VEL
LIN {X 0,Y 397.072,Z 322.021,A -85,B 0,C 180,E1 -11309.117,E2 -11309.117} C_VEL
LIN {X 0,Y 397.093,Z 322.012,A -85,B 0,C 180,E1 -11312.602,E2 -11312.602} C_VEL
LIN {X 0,Y 397.106,Z 322.019,A -85,B 0,C 180,E1 -11315.98,E2 -11315.98} C_VEL
LIN {X 0,Y 397.133,Z 321.994,A -85,B 0,C 180,E1 -11319.704,E2 -11319.704} C_VEL
LIN {X 0,Y 397.176,Z 322.007,A -85,B 0,C 180,E1 -11322.845,E2 -11322.845} C_VEL
LIN {X 0,Y 397.223,Z 321.991,A -85,B 0,C 180,E1 -11326.703,E2 -11326.703} C_VEL
LIN {X 0,Y 397.207,Z 322.009,A -85,B 0,C 180,E1 -11329.809,E2 -11329.809} C_VEL
LIN {X 0,Y 397.322,Z 321.984,A -85,B 0,C 180,E1 -11332.887,E2 -11332.887} C_VEL
LIN {X 0,Y 397.23,Z 321.994,A -85,B 0,C 180,E1 -11334.925,E2 -11334.925} C_VEL
LIN {X 0,Y 397.431,Z 321.978,A -85,B 0,C 180,E1 -11337.973,E2 -11337.973} C_VEL
LIN {X 0,Y 397.435,Z 321.974,A -85,B 0,C 180,E1 -11342.027,E2 -11342.027} C_VEL
LIN {X 0,Y 397.286,Z 321.988,A -85,B 0,C 180,E1 -11346.525,E2 -11346.525} C_VEL
LIN {X 0,Y 397.228,Z 321.995,A -85,B 0,C 180,E1 -11349.163,E2 -11349.163} C_VEL
LIN {X 0,Y 397.211,Z 322.001,A -85,B 0,C 180,E1 -11352.258,E2 -11352.258} C_VEL
LIN {X 0,Y 397.168,Z 322.001,A -85,B 0,C 180,E1 -11355.393,E2 -11355.393} C_VEL
LIN {X 0,Y 397.15,Z 322.01,A -85,B 0,C 180,E1 -11358.574,E2 -11358.574} C_VEL
LIN {X 0,Y 397.088,Z 322.016,A -85,B 0,C 180,E1 -11361.819,E2 -11361.819} C_VEL
LIN {X 0,Y 397.096,Z 322.02,A -85,B 0,C 180,E1 -11365.136,E2 -11365.136} C_VEL
LIN {X 0,Y 397.057,Z 321.997,A -85,B 0,C 180,E1 -11368.549,E2 -11368.549} C_VEL
LIN {X 0,Y 397.075,Z 322.007,A -85,B 0,C 180,E1 -11371.837,E2 -11371.837} C_VEL
LIN {X 0,Y 397.114,Z 322.016,A -85,B 0,C 180,E1 -11374.495,E2 -11374.495} C_VEL
LIN {X 0,Y 397.086,Z 322,A -85,B 0,C 180,E1 -11378.277,E2 -11378.277} C_VEL
LIN {X 0,Y 397.047,Z 322.025,A -85,B 0,C 180,E1 -11381.977,E2 -11381.977} C_VEL
LIN {X 0,Y 397.082,Z 322.017,A -85,B 0,C 180,E1 -11385.07,E2 -11385.07} C_VEL
LIN {X 0,Y 397.048,Z 322.018,A -85,B 0,C 180,E1 -11388.025,E2 -11388.025} C_VEL
LIN {X 0,Y 397.088,Z 322.011,A -85,B 0,C 180,E1 -11391.724,E2 -11391.724} C_VEL
LIN {X 0,Y 397.115,Z 322.02,A -85,B 0,C 180,E1 -11395.506,E2 -11395.506} C_VEL
LIN {X 0,Y 397.073,Z 322.024,A -85,B 0,C 180,E1 -11399.118,E2 -11399.118} C_VEL
LIN {X 0,Y 397.057,Z 321.996,A -85,B 0,C 180,E1 -11402.253,E2 -11402.253} C_VEL
LIN {X 0,Y 397.101,Z 322.02,A -85,B 0,C 180,E1 -11404.865,E2 -11404.865} C_VEL
LIN {X 0,Y 397.095,Z 322.003,A -85,B 0,C 180,E1 -11408.182,E2 -11408.182} C_VEL
LIN {X 0,Y 397.186,Z 322.17,A -85,B 0,C 180,E1 -11410.175,E2 -11410.175} C_VEL
LIN {X 0,Y 397.374,Z 323.066,A -85,B 0,C 180,E1 -11410.341,E2 -11410.341} C_VEL
LIN {X 0,Y 404.141,Z 340.249,A -85,B 0,C 180,E1 -11411.04,E2 -11411.04} C_VEL
LIN {X 0,Y 403.521,Z 401.676,A -85,B 0,C 180,E1 -11412.156,E2 -11412.156} C_VEL
LIN {X 0,Y 403.415,Z 414.268,A -85,B 0,C 180,E1 -11412.544,E2 -11412.544} C_VEL
LIN {X 0,Y 403.085,Z 427.037,A -85,B 0,C 180,E1 -11413.151,E2 -11413.151} C_VEL
LIN {X 0,Y 402.596,Z 438.785,A -85,B 0,C 180,E1 -11413.911,E2 -11413.911} C_VEL
LIN {X 0,Y 401.884,Z 449.467,A -85,B 0,C 180,E1 -11414.793,E2 -11414.793} C_VEL
LIN {X 0,Y 401.107,Z 460.319,A -85,B 0,C 180,E1 -11415.93,E2 -11415.93} C_VEL
LIN {X 0,Y 400.459,Z 469.098,A -85,B 0,C 180,E1 -11417.07,E2 -11417.07} C_VEL
LIN {X 0,Y 399.854,Z 477.132,A -85,B 0,C 180,E1 -11418.339,E2 -11418.339} C_VEL
LIN {X 0,Y 399.132,Z 485.001,A -85,B 0,C 180,E1 -11419.859,E2 -11419.859} C_VEL
LIN {X 0,Y 398.521,Z 490.916,A -85,B 0,C 180,E1 -11421.274,E2 -11421.274} C_VEL
LIN {X 0,Y 398.135,Z 496.297,A -85,B 0,C 180,E1 -11422.902,E2 -11422.902} C_VEL
LIN {X 0,Y 397.618,Z 500.193,A -85,B 0,C 180,E1 -11424.421,E2 -11424.421} C_VEL
LIN {X 0,Y 397.272,Z 503.064,A -85,B 0,C 180,E1 -11425.942,E2 -11425.942} C_VEL
LIN {X 0,Y 397.297,Z 504.414,A -85,B 0,C 180,E1 -11426.958,E2 -11426.958} C_VEL
LIN {X 0,Y 397.136,Z 505.397,A -85,B 0,C 180,E1 -11427.972,E2 -11427.972} C_VEL
LIN {X 0,Y 397.209,Z 505.979,A -85,B 0,C 180,E1 -11428.986,E2 -11428.986} C_VEL
LIN {X 0,Y 397.191,Z 506.209,A -85,B 0,C 180,E1 -11430,E2 -11430} C_VEL
LIN {X 0,Y 397.209,Z 506.024,A -85,B 0,C 180,E1 -11431.014,E2 -11431.014} C_VEL
LIN {X 0,Y 397.136,Z 505.47,A -85,B 0,C 180,E1 -11432.028,E2 -11432.028} C_VEL
LIN {X 0,Y 397.295,Z 504.516,A -85,B 0,C 180,E1 -11433.042,E2 -11433.042} C_VEL
LIN {X 0,Y 397.286,Z 502.927,A -85,B 0,C 180,E1 -11434.221,E2 -11434.221} C_VEL
LIN {X 0,Y 397.672,Z 499.235,A -85,B 0,C 180,E1 -11436.087,E2 -11436.087} C_VEL
LIN {X 0,Y 398.237,Z 495.049,A -85,B 0,C 180,E1 -11437.606,E2 -11437.606} C_VEL
LIN {X 0,Y 398.398,Z 492.521,A -85,B 0,C 180,E1 -11438.376,E2 -11438.376} C_VEL
LIN {X 0,Y 397.976,Z 489.885,A -85,B 0,C 180,E1 -11439.136,E2 -11439.136} C_VEL
LIN {X 0,Y 395.729,Z 485.359,A -85,B 0,C 180,E1 -11440.367,E2 -11440.367} C_VEL
LIN {X 0,Y 393.518,Z 480.207,A -85,B 0,C 180,E1 -11441.553,E2 -11441.553} C_VEL
LIN {X 0,Y 393.146,Z 476.591,A -85,B 0,C 180,E1 -11442.232,E2 -11442.232} C_VEL
LIN {X 0,Y 393.777,Z 468.991,A -85,B 0,C 180,E1 -11443.416,E2 -11443.416} C_VEL
LIN {X 0,Y 394.493,Z 459.959,A -85,B 0,C 180,E1 -11444.574,E2 -11444.574} C_VEL
LIN {X 0,Y 395.32,Z 449.459,A -85,B 0,C 180,E1 -11445.658,E2 -11445.658} C_VEL
LIN {X 0,Y 395.959,Z 437.797,A -85,B 0,C 180,E1 -11446.617,E2 -11446.617} C_VEL
LIN {X 0,Y 396.487,Z 426.36,A -85,B 0,C 180,E1 -11447.338,E2 -11447.338} C_VEL
LIN {X 0,Y 396.716,Z 413.501,A -85,B 0,C 180,E1 -11447.927,E2 -11447.927} C_VEL
LIN {X 0,Y 396.819,Z 399.715,A -85,B 0,C 180,E1 -11448.322,E2 -11448.322} C_VEL
LIN {X 0,Y 397.33,Z 341.193,A -85,B 0,C 180,E1 -11449.4,E2 -11449.4} C_VEL
LIN {X 0,Y 390.319,Z 324.004,A -85,B 0,C 180,E1 -11450.133,E2 -11450.133} C_VEL
LIN {X 0,Y 390.092,Z 323.007,A -85,B 0,C 180,E1 -11450.334,E2 -11450.334} C_VEL
LIN {X 0,Y 390.057,Z 322.883,A -85,B 0,C 180,E1 -11453.352,E2 -11453.352} C_VEL
LIN {X 0,Y 390.025,Z 322.871,A -85,B 0,C 180,E1 -11456.774,E2 -11456.774} C_VEL
LIN {X 0,Y 390.034,Z 322.899,A -85,B 0,C 180,E1 -11460.3,E2 -11460.3} C_VEL
LIN {X 0,Y 390.068,Z 322.893,A -85,B 0,C 180,E1 -11464.024,E2 -11464.024} C_VEL
LIN {X 0,Y 390.034,Z 322.886,A -85,B 0,C 180,E1 -11467.78,E2 -11467.78} C_VEL
LIN {X 0,Y 390.013,Z 322.901,A -85,B 0,C 180,E1 -11470.814,E2 -11470.814} C_VEL
LIN {X 0,Y 390.04,Z 322.881,A -85,B 0,C 180,E1 -11473.884,E2 -11473.884} C_VEL
LIN {X 0,Y 390.043,Z 322.902,A -85,B 0,C 180,E1 -11476.787,E2 -11476.787} C_VEL
LIN {X 0,Y 390.005,Z 322.888,A -85,B 0,C 180,E1 -11479.554,E2 -11479.554} C_VEL
LIN {X 0,Y 390.034,Z 322.882,A -85,B 0,C 180,E1 -11482.45,E2 -11482.45} C_VEL
LIN {X 0,Y 390.064,Z 322.895,A -85,B 0,C 180,E1 -11485.975,E2 -11485.975} C_VEL
LIN {X 0,Y 390.037,Z 322.865,A -85,B 0,C 180,E1 -11489.87,E2 -11489.87} C_VEL
LIN {X 0,Y 390.024,Z 322.892,A -85,B 0,C 180,E1 -11493.225,E2 -11493.225} C_VEL
LIN {X 0,Y 390.052,Z 322.897,A -85,B 0,C 180,E1 -11496.767,E2 -11496.767} C_VEL
LIN {X 0,Y 390.079,Z 322.885,A -85,B 0,C 180,E1 -11499.982,E2 -11499.982} C_VEL
LIN {X 0,Y 390.129,Z 322.884,A -85,B 0,C 180,E1 -11503.248,E2 -11503.248} C_VEL
LIN {X 0,Y 390.189,Z 322.874,A -85,B 0,C 180,E1 -11506.561,E2 -11506.561} C_VEL
LIN {X 0,Y 390.154,Z 322.882,A -85,B 0,C 180,E1 -11509.622,E2 -11509.622} C_VEL
LIN {X 0,Y 390.235,Z 322.866,A -85,B 0,C 180,E1 -11512.758,E2 -11512.758} C_VEL
LIN {X 0,Y 390.192,Z 322.88,A -85,B 0,C 180,E1 -11514.833,E2 -11514.833} C_VEL
LIN {X 0,Y 390.403,Z 322.85,A -85,B 0,C 180,E1 -11517.937,E2 -11517.937} C_VEL
LIN {X 0,Y 390.398,Z 322.854,A -85,B 0,C 180,E1 -11522.063,E2 -11522.063} C_VEL
LIN {X 0,Y 390.295,Z 322.856,A -85,B 0,C 180,E1 -11526.202,E2 -11526.202} C_VEL
LIN {X 0,Y 390.181,Z 322.879,A -85,B 0,C 180,E1 -11529.329,E2 -11529.329} C_VEL
LIN {X 0,Y 390.188,Z 322.868,A -85,B 0,C 180,E1 -11533.439,E2 -11533.439} C_VEL
LIN {X 0,Y 390.123,Z 322.885,A -85,B 0,C 180,E1 -11537.298,E2 -11537.298} C_VEL
LIN {X 0,Y 390.081,Z 322.871,A -85,B 0,C 180,E1 -11540.47,E2 -11540.47} C_VEL
LIN {X 0,Y 390.056,Z 322.892,A -85,B 0,C 180,E1 -11543.353,E2 -11543.353} C_VEL
LIN {X 0,Y 390.042,Z 322.89,A -85,B 0,C 180,E1 -11546.774,E2 -11546.774} C_VEL
LIN {X 0,Y 390.032,Z 322.898,A -85,B 0,C 180,E1 -11550.3,E2 -11550.3} C_VEL
LIN {X 0,Y 390.064,Z 322.887,A -85,B 0,C 180,E1 -11554.025,E2 -11554.025} C_VEL
LIN {X 0,Y 390.031,Z 322.903,A -85,B 0,C 180,E1 -11557.781,E2 -11557.781} C_VEL
LIN {X 0,Y 390.012,Z 322.902,A -85,B 0,C 180,E1 -11560.815,E2 -11560.815} C_VEL
LIN {X 0,Y 390.04,Z 322.878,A -85,B 0,C 180,E1 -11563.885,E2 -11563.885} C_VEL
LIN {X 0,Y 390.043,Z 322.893,A -85,B 0,C 180,E1 -11566.789,E2 -11566.789} C_VEL
LIN {X 0,Y 390.006,Z 322.892,A -85,B 0,C 180,E1 -11569.555,E2 -11569.555} C_VEL
LIN {X 0,Y 390.035,Z 322.903,A -85,B 0,C 180,E1 -11572.451,E2 -11572.451} C_VEL
LIN {X 0,Y 390.06,Z 322.897,A -85,B 0,C 180,E1 -11576.045,E2 -11576.045} C_VEL
LIN {X 0,Y 390.123,Z 323.169,A -85,B 0,C 180,E1 -11576.536,E2 -11576.536} C_VEL
LIN {X 0,Y 393.501,Z 337.48,A -85,B 0,C 180,E1 -11579.291,E2 -11579.291} C_VEL
LIN {X 0,Y 395.26,Z 346.001,A -85,B 0,C 180,E1 -11580.851,E2 -11580.851} C_VEL
LIN {X 0,Y 395.101,Z 350.425,A -85,B 0,C 180,E1 -11581.587,E2 -11581.587} C_VEL
LIN {X 0,Y 393.748,Z 367.424,A -85,B 0,C 180,E1 -11584.353,E2 -11584.353} C_VEL
LIN {X 0,Y 392.44,Z 385.901,A -85,B 0,C 180,E1 -11587.355,E2 -11587.355} C_VEL
LIN {X 0,Y 391.584,Z 398.864,A -85,B 0,C 180,E1 -11589.446,E2 -11589.446} C_VEL
LIN {X 0,Y 394.575,Z 424.299,A -85,B 0,C 180,E1 -11590.113,E2 -11590.113} C_VEL
LIN {X 0,Y 396.309,Z 443.777,A -85,B 0,C 180,E1 -11590.564,E2 -11590.564} C_VEL
LIN {X 0,Y 395.372,Z 509.654,A -85,B 0,C 180,E1 -11591.776,E2 -11591.776} C_VEL
LIN {X 0,Y 394.825,Z 522.948,A -85,B 0,C 180,E1 -11592.219,E2 -11592.219} C_VEL
LIN {X 0,Y 393.886,Z 536.276,A -85,B 0,C 180,E1 -11592.878,E2 -11592.878} C_VEL
LIN {X 0,Y 392.961,Z 547.499,A -85,B 0,C 180,E1 -11593.64,E2 -11593.64} C_VEL
LIN {X 0,Y 391.919,Z 559.205,A -85,B 0,C 180,E1 -11594.663,E2 -11594.663} C_VEL
LIN {X 0,Y 391.051,Z 569.685,A -85,B 0,C 180,E1 -11595.813,E2 -11595.813} C_VEL
LIN {X 0,Y 390.52,Z 578.499,A -85,B 0,C 180,E1 -11597,E2 -11597} C_VEL
LIN {X 0,Y 389.807,Z 586.523,A -85,B 0,C 180,E1 -11598.298,E2 -11598.298} C_VEL
LIN {X 0,Y 389.339,Z 594.412,A -85,B 0,C 180,E1 -11599.863,E2 -11599.863} C_VEL
LIN {X 0,Y 389.205,Z 601.737,A -85,B 0,C 180,E1 -11601.694,E2 -11601.694} C_VEL
LIN {X 0,Y 389.23,Z 606.636,A -85,B 0,C 180,E1 -11603.261,E2 -11603.261} C_VEL
LIN {X 0,Y 389.321,Z 610.389,A -85,B 0,C 180,E1 -11604.822,E2 -11604.822} C_VEL
LIN {X 0,Y 389.485,Z 612.342,A -85,B 0,C 180,E1 -11605.861,E2 -11605.861} C_VEL
LIN {X 0,Y 389.503,Z 613.794,A -85,B 0,C 180,E1 -11606.897,E2 -11606.897} C_VEL
LIN {X 0,Y 389.825,Z 615.503,A -85,B 0,C 180,E1 -11608.967,E2 -11608.967} C_VEL
LIN {X 0,Y 389.859,Z 615.73,A -85,B 0,C 180,E1 -11610,E2 -11610} C_VEL
LIN {X 0,Y 389.825,Z 615.5,A -85,B 0,C 180,E1 -11611.033,E2 -11611.033} C_VEL
LIN {X 0,Y 389.503,Z 613.79,A -85,B 0,C 180,E1 -11613.103,E2 -11613.103} C_VEL
LIN {X 0,Y 389.501,Z 612.338,A -85,B 0,C 180,E1 -11614.139,E2 -11614.139} C_VEL
LIN {X 0,Y 389.279,Z 609.26,A -85,B 0,C 180,E1 -11615.699,E2 -11615.699} C_VEL
LIN {X 0,Y 389.222,Z 605.128,A -85,B 0,C 180,E1 -11617.261,E2 -11617.261} C_VEL
LIN {X 0,Y 389.208,Z 598.79,A -85,B 0,C 180,E1 -11619.091,E2 -11619.091} C_VEL
LIN {X 0,Y 389.501,Z 591.92,A -85,B 0,C 180,E1 -11620.658,E2 -11620.658} C_VEL
LIN {X 0,Y 389.955,Z 583.428,A -85,B 0,C 180,E1 -11622.226,E2 -11622.226} C_VEL
LIN {X 0,Y 390.554,Z 576.613,A -85,B 0,C 180,E1 -11623.264,E2 -11623.264} C_VEL
LIN {X 0,Y 391.313,Z 566.46,A -85,B 0,C 180,E1 -11624.562,E2 -11624.562} C_VEL
LIN {X 0,Y 392.17,Z 556.483,A -85,B 0,C 180,E1 -11625.593,E2 -11625.593} C_VEL
LIN {X 0,Y 393.106,Z 545.684,A -85,B 0,C 180,E1 -11626.488,E2 -11626.488} C_VEL
LIN {X 0,Y 394.143,Z 532.721,A -85,B 0,C 180,E1 -11627.311,E2 -11627.311} C_VEL
LIN {X 0,Y 394.993,Z 519.571,A -85,B 0,C 180,E1 -11627.907,E2 -11627.907} C_VEL
LIN {X 0,Y 395.439,Z 506.435,A -85,B 0,C 180,E1 -11628.288,E2 -11628.288} C_VEL
LIN {X 0,Y 396.167,Z 440.775,A -85,B 0,C 180,E1 -11629.49,E2 -11629.49} C_VEL
LIN {X 0,Y 392.05,Z 402.827,A -85,B 0,C 180,E1 -11630.412,E2 -11630.412} C_VEL
LIN {X 0,Y 391.584,Z 398.792,A -85,B 0,C 180,E1 -11630.554,E2 -11630.554} C_VEL
LIN {X 0,Y 393.117,Z 375.778,A -85,B 0,C 180,E1 -11634.279,E2 -11634.279} C_VEL
LIN {X 0,Y 394.694,Z 355.47,A -85,B 0,C 180,E1 -11637.578,E2 -11637.578} C_VEL
LIN {X 0,Y 395.374,Z 347.31,A -85,B 0,C 180,E1 -11638.907,E2 -11638.907} C_VEL
LIN {X 0,Y 393.764,Z 338.564,A -85,B 0,C 180,E1 -11640.493,E2 -11640.493} C_VEL
LIN {X 0,Y 390.256,Z 323.79,A -85,B 0,C 180,E1 -11643.316,E2 -11643.316} C_VEL
LIN {X 0,Y 390.069,Z 322.948,A -85,B 0,C 180,E1 -11643.566,E2 -11643.566} C_VEL
LIN {X 0,Y 390.047,Z 322.892,A -85,B 0,C 180,E1 -11646.484,E2 -11646.484} C_VEL
LIN {X 0,Y 390.033,Z 322.885,A -85,B 0,C 180,E1 -11649.211,E2 -11649.211} C_VEL
LIN {X 0,Y 390.026,Z 322.902,A -85,B 0,C 180,E1 -11652.371,E2 -11652.371} C_VEL
LIN {X 0,Y 390.036,Z 322.872,A -85,B 0,C 180,E1 -11655.353,E2 -11655.353} C_VEL
LIN {X 0,Y 390.011,Z 322.906,A -85,B 0,C 180,E1 -11658.184,E2 -11658.184} C_VEL
LIN {X 0,Y 390.052,Z 322.879,A -85,B 0,C 180,E1 -11660.903,E2 -11660.903} C_VEL
LIN {X 0,Y 390.063,Z 322.872,A -85,B 0,C 180,E1 -11664.791,E2 -11664.791} C_VEL
LIN {X 0,Y 390.017,Z 322.901,A -85,B 0,C 180,E1 -11668.495,E2 -11668.495} C_VEL
LIN {X 0,Y 390.031,Z 322.887,A -85,B 0,C 180,E1 -11672.063,E2 -11672.063} C_VEL
LIN {X 0,Y 390.037,Z 322.901,A -85,B 0,C 180,E1 -11675.516,E2 -11675.516} C_VEL
LIN {X 0,Y 390.049,Z 322.876,A -85,B 0,C 180,E1 -11678.877,E2 -11678.877} C_VEL
LIN {X 0,Y 390.121,Z 322.889,A -85,B 0,C 180,E1 -11682.166,E2 -11682.166} C_VEL
LIN {X 0,Y 390.137,Z 322.887,A -85,B 0,C 180,E1 -11685.392,E2 -11685.392} C_VEL
LIN {X 0,Y 390.138,Z 322.882,A -85,B 0,C 180,E1 -11688.571,E2 -11688.571} C_VEL
LIN {X 0,Y 390.263,Z 322.866,A -85,B 0,C 180,E1 -11692.072,E2 -11692.072} C_VEL
LIN {X 0,Y 390.202,Z 322.869,A -85,B 0,C 180,E1 -11694.833,E2 -11694.833} C_VEL
LIN {X 0,Y 390.398,Z 322.854,A -85,B 0,C 180,E1 -11697.937,E2 -11697.937} C_VEL
LIN {X 0,Y 390.403,Z 322.85,A -85,B 0,C 180,E1 -11702.063,E2 -11702.063} C_VEL
LIN {X 0,Y 390.246,Z 322.864,A -85,B 0,C 180,E1 -11706.517,E2 -11706.517} C_VEL
LIN {X 0,Y 390.185,Z 322.873,A -85,B 0,C 180,E1 -11709.329,E2 -11709.329} C_VEL
LIN {X 0,Y 390.163,Z 322.878,A -85,B 0,C 180,E1 -11712.483,E2 -11712.483} C_VEL
LIN {X 0,Y 390.129,Z 322.881,A -85,B 0,C 180,E1 -11715.677,E2 -11715.677} C_VEL
LIN {X 0,Y 390.095,Z 322.89,A -85,B 0,C 180,E1 -11718.923,E2 -11718.923} C_VEL
LIN {X 0,Y 390.028,Z 322.897,A -85,B 0,C 180,E1 -11722.235,E2 -11722.235} C_VEL
LIN {X 0,Y 390.044,Z 322.893,A -85,B 0,C 180,E1 -11725.723,E2 -11725.723} C_VEL
LIN {X 0,Y 390.017,Z 322.866,A -85,B 0,C 180,E1 -11729.113,E2 -11729.113} C_VEL
LIN {X 0,Y 390.036,Z 322.891,A -85,B 0,C 180,E1 -11732.722,E2 -11732.722} C_VEL
LIN {X 0,Y 390.048,Z 322.895,A -85,B 0,C 180,E1 -11735.825,E2 -11735.825} C_VEL
LIN {X 0,Y 390.032,Z 322.873,A -85,B 0,C 180,E1 -11739.213,E2 -11739.213} C_VEL
LIN {X 0,Y 390.026,Z 322.898,A -85,B 0,C 180,E1 -11742.373,E2 -11742.373} C_VEL
LIN {X 0,Y 390.037,Z 322.889,A -85,B 0,C 180,E1 -11745.354,E2 -11745.354} C_VEL
LIN {X 0,Y 390.011,Z 322.896,A -85,B 0,C 180,E1 -11748.185,E2 -11748.185} C_VEL
LIN {X 0,Y 390.055,Z 322.898,A -85,B 0,C 180,E1 -11750.904,E2 -11750.904} C_VEL
LIN {X 0,Y 390.067,Z 322.895,A -85,B 0,C 180,E1 -11754.792,E2 -11754.792} C_VEL
LIN {X 0,Y 390.018,Z 322.899,A -85,B 0,C 180,E1 -11758.496,E2 -11758.496} C_VEL
LIN {X 0,Y 390.015,Z 322.874,A -85,B 0,C 180,E1 -11762.004,E2 -11762.004} C_VEL
LIN {X 0,Y 390.042,Z 322.904,A -85,B 0,C 180,E1 -11765.517,E2 -11765.517} C_VEL
LIN {X 0,Y 390.061,Z 322.886,A -85,B 0,C 180,E1 -11768.879,E2 -11768.879} C_VEL
LIN {X 0,Y 390.159,Z 323.172,A -85,B 0,C 180,E1 -11769.843,E2 -11769.843} C_VEL
LIN {X 0,Y 390.432,Z 324.251,A -85,B 0,C 180,E1 -11769.988,E2 -11769.988} C_VEL
LIN {X 0,Y 397.378,Z 341.34,A -85,B 0,C 180,E1 -11770.706,E2 -11770.706} C_VEL
LIN {X 0,Y 396.829,Z 404.143,A -85,B 0,C 180,E1 -11771.879,E2 -11771.879} C_VEL
LIN {X 0,Y 396.638,Z 416.802,A -85,B 0,C 180,E1 -11772.303,E2 -11772.303} C_VEL
LIN {X 0,Y 396.3,Z 429.144,A -85,B 0,C 180,E1 -11772.92,E2 -11772.92} C_VEL
LIN {X 0,Y 395.794,Z 441.483,A -85,B 0,C 180,E1 -11773.758,E2 -11773.758} C_VEL
LIN {X 0,Y 394.94,Z 453.062,A -85,B 0,C 180,E1 -11774.783,E2 -11774.783} C_VEL
LIN {X 0,Y 394.158,Z 463.396,A -85,B 0,C 180,E1 -11775.94,E2 -11775.94} C_VEL
LIN {X 0,Y 393.496,Z 471.82,A -85,B 0,C 180,E1 -11777.1,E2 -11777.1} C_VEL
LIN {X 0,Y 392.771,Z 479.575,A -85,B 0,C 180,E1 -11778.387,E2 -11778.387} C_VEL
LIN {X 0,Y 392.055,Z 487.251,A -85,B 0,C 180,E1 -11779.96,E2 -11779.96} C_VEL
LIN {X 0,Y 391.504,Z 493.005,A -85,B 0,C 180,E1 -11781.43,E2 -11781.43} C_VEL
LIN {X 0,Y 391.163,Z 497.277,A -85,B 0,C 180,E1 -11782.775,E2 -11782.775} C_VEL
LIN {X 0,Y 390.623,Z 501.173,A -85,B 0,C 180,E1 -11784.321,E2 -11784.321} C_VEL
LIN {X 0,Y 390.258,Z 504.043,A -85,B 0,C 180,E1 -11785.869,E2 -11785.869} C_VEL
LIN {X 0,Y 390.279,Z 505.392,A -85,B 0,C 180,E1 -11786.903,E2 -11786.903} C_VEL
LIN {X 0,Y 390.114,Z 506.375,A -85,B 0,C 180,E1 -11787.935,E2 -11787.935} C_VEL
LIN {X 0,Y 390.184,Z 506.957,A -85,B 0,C 180,E1 -11788.968,E2 -11788.968} C_VEL
LIN {X 0,Y 390.167,Z 507.186,A -85,B 0,C 180,E1 -11790,E2 -11790} C_VEL
LIN {X 0,Y 390.184,Z 507.002,A -85,B 0,C 180,E1 -11791.032,E2 -11791.032} C_VEL
LIN {X 0,Y 390.114,Z 506.448,A -85,B 0,C 180,E1 -11792.065,E2 -11792.065} C_VEL
LIN {X 0,Y 390.276,Z 505.494,A -85,B 0,C 180,E1 -11793.097,E2 -11793.097} C_VEL
LIN {X 0,Y 390.249,Z 504.191,A -85,B 0,C 180,E1 -11794.131,E2 -11794.131} C_VEL
LIN {X 0,Y 390.619,Z 501.375,A -85,B 0,C 180,E1 -11795.679,E2 -11795.679} C_VEL
LIN {X 0,Y 391.14,Z 497.55,A -85,B 0,C 180,E1 -11797.225,E2 -11797.225} C_VEL
LIN {X 0,Y 391.519,Z 492.473,A -85,B 0,C 180,E1 -11798.828,E2 -11798.828} C_VEL
LIN {X 0,Y 392.31,Z 485.239,A -85,B 0,C 180,E1 -11800.581,E2 -11800.581} C_VEL
LIN {X 0,Y 393.112,Z 477.211,A -85,B 0,C 180,E1 -11802.126,E2 -11802.126} C_VEL
LIN {X 0,Y 393.146,Z 476.591,A -85,B 0,C 180,E1 -11802.232,E2 -11802.232} C_VEL
LIN {X 0,Y 392.763,Z 472.81,A -85,B 0,C 180,E1 -11802.889,E2 -11802.889} C_VEL
LIN {X 0,Y 390.551,Z 466.454,A -85,B 0,C 180,E1 -11803.958,E2 -11803.958} C_VEL
LIN {X 0,Y 388.434,Z 459.601,A -85,B 0,C 180,E1 -11804.955,E2 -11804.955} C_VEL
LIN {X 0,Y 388.183,Z 454.98,A -85,B 0,C 180,E1 -11805.49,E2 -11805.49} C_VEL
LIN {X 0,Y 388.955,Z 443.987,A -85,B 0,C 180,E1 -11806.507,E2 -11806.507} C_VEL
LIN {X 0,Y 389.592,Z 431.807,A -85,B 0,C 180,E1 -11807.383,E2 -11807.383} C_VEL
LIN {X 0,Y 389.986,Z 419.298,A -85,B 0,C 180,E1 -11808.043,E2 -11808.043} C_VEL
LIN {X 0,Y 390.129,Z 407.445,A -85,B 0,C 180,E1 -11808.478,E2 -11808.478} C_VEL
LIN {X 0,Y 390.172,Z 386.581,A -85,B 0,C 180,E1 -11808.918,E2 -11808.918} C_VEL
LIN {X 0,Y 390.671,Z 342.896,A -85,B 0,C 180,E1 -11809.73,E2 -11809.73} C_VEL
LIN {X 0,Y 383.625,Z 325.853,A -85,B 0,C 180,E1 -11810.466,E2 -11810.466} C_VEL
LIN {X 0,Y 383.085,Z 324.207,A -85,B 0,C 180,E1 -11810.616,E2 -11810.616} C_VEL
LIN {X 0,Y 383.031,Z 323.835,A -85,B 0,C 180,E1 -11810.768,E2 -11810.768} C_VEL
LIN {X 0,Y 383.008,Z 323.768,A -85,B 0,C 180,E1 -11813.809,E2 -11813.809} C_VEL
LIN {X 0,Y 382.965,Z 323.746,A -85,B 0,C 180,E1 -11817.308,E2 -11817.308} C_VEL
LIN {X 0,Y 382.977,Z 323.78,A -85,B 0,C 180,E1 -11820.918,E2 -11820.918} C_VEL
LIN {X 0,Y 383.009,Z 323.778,A -85,B 0,C 180,E1 -11824.668,E2 -11824.668} C_VEL
LIN {X 0,Y 382.99,Z 323.764,A -85,B 0,C 180,E1 -11827.901,E2 -11827.901} C_VEL
LIN {X 0,Y 382.957,Z 323.776,A -85,B 0,C 180,E1 -11831.35,E2 -11831.35} C_VEL
LIN {X 0,Y 382.985,Z 323.762,A -85,B 0,C 180,E1 -11834.301,E2 -11834.301} C_VEL
LIN {X 0,Y 382.978,Z 323.778,A -85,B 0,C 180,E1 -11837.235,E2 -11837.235} C_VEL
LIN {X 0,Y 382.981,Z 323.753,A -85,B 0,C 180,E1 -11840.418,E2 -11840.418} C_VEL
LIN {X 0,Y 383.018,Z 323.769,A -85,B 0,C 180,E1 -11844.043,E2 -11844.043} C_VEL
LIN {X 0,Y 382.98,Z 323.769,A -85,B 0,C 180,E1 -11847.578,E2 -11847.578} C_VEL
LIN {X 0,Y 382.969,Z 323.742,A -85,B 0,C 180,E1 -11850.298,E2 -11850.298} C_VEL
LIN {X 0,Y 382.997,Z 323.768,A -85,B 0,C 180,E1 -11854.045,E2 -11854.045} C_VEL
LIN {X 0,Y 382.979,Z 323.774,A -85,B 0,C 180,E1 -11857.333,E2 -11857.333} C_VEL
LIN {X 0,Y 383.042,Z 323.77,A -85,B 0,C 180,E1 -11860.715,E2 -11860.715} C_VEL
LIN {X 0,Y 383.068,Z 323.766,A -85,B 0,C 180,E1 -11864.026,E2 -11864.026} C_VEL
LIN {X 0,Y 383.129,Z 323.756,A -85,B 0,C 180,E1 -11867.284,E2 -11867.284} C_VEL
LIN {X 0,Y 383.131,Z 323.755,A -85,B 0,C 180,E1 -11870.497,E2 -11870.497} C_VEL
LIN {X 0,Y 383.222,Z 323.741,A -85,B 0,C 180,E1 -11873.683,E2 -11873.683} C_VEL
LIN {X 0,Y 383.369,Z 323.726,A -85,B 0,C 180,E1 -11877.899,E2 -11877.899} C_VEL
LIN {X 0,Y 383.364,Z 323.73,A -85,B 0,C 180,E1 -11882.101,E2 -11882.101} C_VEL
LIN {X 0,Y 383.252,Z 323.733,A -85,B 0,C 180,E1 -11886.317,E2 -11886.317} C_VEL
LIN {X 0,Y 383.131,Z 323.757,A -85,B 0,C 180,E1 -11889.503,E2 -11889.503} C_VEL
LIN {X 0,Y 383.119,Z 323.749,A -85,B 0,C 180,E1 -11893.536,E2 -11893.536} C_VEL
LIN {X 0,Y 383.088,Z 323.762,A -85,B 0,C 180,E1 -11897.069,E2 -11897.069} C_VEL
LIN {X 0,Y 383.022,Z 323.75,A -85,B 0,C 180,E1 -11900.647,E2 -11900.647} C_VEL
LIN {X 0,Y 383.004,Z 323.773,A -85,B 0,C 180,E1 -11903.809,E2 -11903.809} C_VEL
LIN {X 0,Y 382.981,Z 323.768,A -85,B 0,C 180,E1 -11907.308,E2 -11907.308} C_VEL
LIN {X 0,Y 382.976,Z 323.778,A -85,B 0,C 180,E1 -11910.919,E2 -11910.919} C_VEL
LIN {X 0,Y 383.006,Z 323.764,A -85,B 0,C 180,E1 -11914.669,E2 -11914.669} C_VEL
LIN {X 0,Y 382.987,Z 323.779,A -85,B 0,C 180,E1 -11917.903,E2 -11917.903} C_VEL
LIN {X 0,Y 382.956,Z 323.781,A -85,B 0,C 180,E1 -11921.351,E2 -11921.351} C_VEL
LIN {X 0,Y 382.984,Z 323.751,A -85,B 0,C 180,E1 -11924.303,E2 -11924.303} C_VEL
LIN {X 0,Y 382.979,Z 323.776,A -85,B 0,C 180,E1 -11927.237,E2 -11927.237} C_VEL
LIN {X 0,Y 382.982,Z 323.761,A -85,B 0,C 180,E1 -11930.42,E2 -11930.42} C_VEL
LIN {X 0,Y 383.01,Z 323.763,A -85,B 0,C 180,E1 -11934.044,E2 -11934.044} C_VEL
LIN {X 0,Y 383.058,Z 324.002,A -85,B 0,C 180,E1 -11936.161,E2 -11936.161} C_VEL
LIN {X 0,Y 386.494,Z 338.425,A -85,B 0,C 180,E1 -11939.007,E2 -11939.007} C_VEL
LIN {X 0,Y 388.434,Z 347.781,A -85,B 0,C 180,E1 -11940.757,E2 -11940.757} C_VEL
LIN {X 0,Y 387.32,Z 363.099,A -85,B 0,C 180,E1 -11943.315,E2 -11943.315} C_VEL
LIN {X 0,Y 385.561,Z 384.917,A -85,B 0,C 180,E1 -11946.928,E2 -11946.928} C_VEL
LIN {X 0,Y 384.673,Z 397.979,A -85,B 0,C 180,E1 -11949.07,E2 -11949.07} C_VEL
LIN {X 0,Y 387.879,Z 424.857,A -85,B 0,C 180,E1 -11949.784,E2 -11949.784} C_VEL
LIN {X 0,Y 389.583,Z 443.614,A -85,B 0,C 180,E1 -11950.23,E2 -11950.23} C_VEL
LIN {X 0,Y 388.63,Z 508.678,A -85,B 0,C 180,E1 -11951.448,E2 -11951.448} C_VEL
LIN {X 0,Y 388.05,Z 521.966,A -85,B 0,C 180,E1 -11951.898,E2 -11951.898} C_VEL
LIN {X 0,Y 387.088,Z 535.292,A -85,B 0,C 180,E1 -11952.568,E2 -11952.568} C_VEL
LIN {X 0,Y 386.116,Z 546.51,A -85,B 0,C 180,E1 -11953.341,E2 -11953.341} C_VEL
LIN {X 0,Y 385.002,Z 558.21,A -85,B 0,C 180,E1 -11954.38,E2 -11954.38} C_VEL
LIN {X 0,Y 384.09,Z 568.798,A -85,B 0,C 180,E1 -11955.564,E2 -11955.564} C_VEL
LIN {X 0,Y 383.509,Z 577.5,A -85,B 0,C 180,E1 -11956.758,E2 -11956.758} C_VEL
LIN {X 0,Y 382.776,Z 585.526,A -85,B 0,C 180,E1 -11958.08,E2 -11958.08} C_VEL
LIN {X 0,Y 382.297,Z 593.418,A -85,B 0,C 180,E1 -11959.675,E2 -11959.675} C_VEL
LIN {X 0,Y 382.12,Z 600.741,A -85,B 0,C 180,E1 -11961.539,E2 -11961.539} C_VEL
LIN {X 0,Y 382.16,Z 605.971,A -85,B 0,C 180,E1 -11963.252,E2 -11963.252} C_VEL
LIN {X 0,Y 382.242,Z 609.4,A -85,B 0,C 180,E1 -11964.725,E2 -11964.725} C_VEL
LIN {X 0,Y 382.409,Z 611.356,A -85,B 0,C 180,E1 -11965.784,E2 -11965.784} C_VEL
LIN {X 0,Y 382.452,Z 612.812,A -85,B 0,C 180,E1 -11966.84,E2 -11966.84} C_VEL
LIN {X 0,Y 382.793,Z 614.524,A -85,B 0,C 180,E1 -11968.948,E2 -11968.948} C_VEL
LIN {X 0,Y 382.834,Z 614.753,A -85,B 0,C 180,E1 -11970,E2 -11970} C_VEL
LIN {X 0,Y 382.793,Z 614.521,A -85,B 0,C 180,E1 -11971.052,E2 -11971.052} C_VEL
LIN {X 0,Y 382.454,Z 612.807,A -85,B 0,C 180,E1 -11973.16,E2 -11973.16} C_VEL
LIN {X 0,Y 382.424,Z 611.35,A -85,B 0,C 180,E1 -11974.216,E2 -11974.216} C_VEL
LIN {X 0,Y 382.219,Z 608.271,A -85,B 0,C 180,E1 -11975.804,E2 -11975.804} C_VEL
LIN {X 0,Y 382.134,Z 604.133,A -85,B 0,C 180,E1 -11977.397,E2 -11977.397} C_VEL
LIN {X 0,Y 382.154,Z 597.794,A -85,B 0,C 180,E1 -11979.26,E2 -11979.26} C_VEL
LIN {X 0,Y 382.472,Z 590.923,A -85,B 0,C 180,E1 -11980.856,E2 -11980.856} C_VEL
LIN {X 0,Y 382.978,Z 582.432,A -85,B 0,C 180,E1 -11982.452,E2 -11982.452} C_VEL
LIN {X 0,Y 383.651,Z 573.765,A -85,B 0,C 180,E1 -11983.777,E2 -11983.777} C_VEL
LIN {X 0,Y 384.567,Z 563.104,A -85,B 0,C 180,E1 -11985.095,E2 -11985.095} C_VEL
LIN {X 0,Y 385.438,Z 554.048,A -85,B 0,C 180,E1 -11986.009,E2 -11986.009} C_VEL
LIN {X 0,Y 386.431,Z 542.905,A -85,B 0,C 180,E1 -11986.917,E2 -11986.917} C_VEL
LIN {X 0,Y 387.458,Z 530.59,A -85,B 0,C 180,E1 -11987.687,E2 -11987.687} C_VEL
LIN {X 0,Y 388.272,Z 517.653,A -85,B 0,C 180,E1 -11988.262,E2 -11988.262} C_VEL
LIN {X 0,Y 388.716,Z 503.918,A -85,B 0,C 180,E1 -11988.65,E2 -11988.65} C_VEL
LIN {X 0,Y 389.536,Z 442.613,A -85,B 0,C 180,E1 -11989.781,E2 -11989.781} C_VEL
LIN {X 0,Y 385.729,Z 406.617,A -85,B 0,C 180,E1 -11990.669,E2 -11990.669} C_VEL
LIN {X 0,Y 384.667,Z 397.888,A -85,B 0,C 180,E1 -11990.928,E2 -11990.928} C_VEL
LIN {X 0,Y 386.198,Z 376.174,A -85,B 0,C 180,E1 -11994.509,E2 -11994.509} C_VEL
LIN {X 0,Y 387.953,Z 354.526,A -85,B 0,C 180,E1 -11998.099,E2 -11998.099} C_VEL
LIN {X 0,Y 388.431,Z 347.707,A -85,B 0,C 180,E1 -11999.243,E2 -11999.243} C_VEL
LIN {X 0,Y 385.399,Z 333.503,A -85,B 0,C 180,E1 -12001.926,E2 -12001.926} C_VEL
LIN {X 0,Y 383.04,Z 323.875,A -85,B 0,C 180,E1 -12003.88,E2 -12003.88} C_VEL
LIN {X 0,Y 382.987,Z 323.78,A -85,B 0,C 180,E1 -12007.269,E2 -12007.269} C_VEL
LIN {X 0,Y 382.971,Z 323.764,A -85,B 0,C 180,E1 -12009.962,E2 -12009.962} C_VEL
LIN {X 0,Y 383.003,Z 323.774,A -85,B 0,C 180,E1 -12012.778,E2 -12012.778} C_VEL
LIN {X 0,Y 382.986,Z 323.753,A -85,B 0,C 180,E1 -12015.787,E2 -12015.787} C_VEL
LIN {X 0,Y 382.957,Z 323.781,A -85,B 0,C 180,E1 -12018.8,E2 -12018.8} C_VEL
LIN {X 0,Y 382.987,Z 323.733,A -85,B 0,C 180,E1 -12022.097,E2 -12022.097} C_VEL
LIN {X 0,Y 383.006,Z 323.755,A -85,B 0,C 180,E1 -12025.331,E2 -12025.331} C_VEL
LIN {X 0,Y 382.976,Z 323.777,A -85,B 0,C 180,E1 -12029.081,E2 -12029.081} C_VEL
LIN {X 0,Y 382.985,Z 323.769,A -85,B 0,C 180,E1 -12032.693,E2 -12032.693} C_VEL
LIN {X 0,Y 383.004,Z 323.773,A -85,B 0,C 180,E1 -12036.191,E2 -12036.191} C_VEL
LIN {X 0,Y 383.049,Z 323.747,A -85,B 0,C 180,E1 -12039.598,E2 -12039.598} C_VEL
LIN {X 0,Y 383.099,Z 323.761,A -85,B 0,C 180,E1 -12042.931,E2 -12042.931} C_VEL
LIN {X 0,Y 383.119,Z 323.748,A -85,B 0,C 180,E1 -12046.464,E2 -12046.464} C_VEL
LIN {X 0,Y 383.135,Z 323.758,A -85,B 0,C 180,E1 -12050.498,E2 -12050.498} C_VEL
LIN {X 0,Y 383.252,Z 323.734,A -85,B 0,C 180,E1 -12053.683,E2 -12053.683} C_VEL
LIN {X 0,Y 383.365,Z 323.731,A -85,B 0,C 180,E1 -12057.899,E2 -12057.899} C_VEL
LIN {X 0,Y 383.369,Z 323.726,A -85,B 0,C 180,E1 -12062.101,E2 -12062.101} C_VEL
LIN {X 0,Y 383.21,Z 323.74,A -85,B 0,C 180,E1 -12066.506,E2 -12066.506} C_VEL
LIN {X 0,Y 383.135,Z 323.753,A -85,B 0,C 180,E1 -12069.503,E2 -12069.503} C_VEL
LIN {X 0,Y 383.119,Z 323.752,A -85,B 0,C 180,E1 -12073.536,E2 -12073.536} C_VEL
LIN {X 0,Y 383.07,Z 323.768,A -85,B 0,C 180,E1 -12077.446,E2 -12077.446} C_VEL
LIN {X 0,Y 383.023,Z 323.761,A -85,B 0,C 180,E1 -12080.647,E2 -12080.647} C_VEL
LIN {X 0,Y 383.004,Z 323.777,A -85,B 0,C 180,E1 -12083.809,E2 -12083.809} C_VEL
LIN {X 0,Y 382.963,Z 323.762,A -85,B 0,C 180,E1 -12087.309,E2 -12087.309} C_VEL
LIN {X 0,Y 382.975,Z 323.75,A -85,B 0,C 180,E1 -12090.919,E2 -12090.919} C_VEL
LIN {X 0,Y 383.012,Z 323.773,A -85,B 0,C 180,E1 -12094.669,E2 -12094.669} C_VEL
LIN {X 0,Y 382.988,Z 323.757,A -85,B 0,C 180,E1 -12097.903,E2 -12097.903} C_VEL
LIN {X 0,Y 382.956,Z 323.771,A -85,B 0,C 180,E1 -12101.351,E2 -12101.351} C_VEL
LIN {X 0,Y 382.986,Z 323.775,A -85,B 0,C 180,E1 -12104.303,E2 -12104.303} C_VEL
LIN {X 0,Y 382.979,Z 323.759,A -85,B 0,C 180,E1 -12107.237,E2 -12107.237} C_VEL
LIN {X 0,Y 382.983,Z 323.777,A -85,B 0,C 180,E1 -12110.42,E2 -12110.42} C_VEL
LIN {X 0,Y 383.012,Z 323.772,A -85,B 0,C 180,E1 -12114.044,E2 -12114.044} C_VEL
LIN {X 0,Y 382.982,Z 323.77,A -85,B 0,C 180,E1 -12117.58,E2 -12117.58} C_VEL
LIN {X 0,Y 382.974,Z 323.777,A -85,B 0,C 180,E1 -12120.299,E2 -12120.299} C_VEL
LIN {X 0,Y 383.002,Z 323.757,A -85,B 0,C 180,E1 -12124.046,E2 -12124.046} C_VEL
LIN {X 0,Y 382.986,Z 323.759,A -85,B 0,C 180,E1 -12127.334,E2 -12127.334} C_VEL
LIN {X 0,Y 383.088,Z 324.04,A -85,B 0,C 180,E1 -12129.444,E2 -12129.444} C_VEL
LIN {X 0,Y 383.369,Z 325.082,A -85,B 0,C 180,E1 -12129.597,E2 -12129.597} C_VEL
LIN {X 0,Y 390.704,Z 343.046,A -85,B 0,C 180,E1 -12130.376,E2 -12130.376} C_VEL
LIN {X 0,Y 390.133,Z 405.281,A -85,B 0,C 180,E1 -12131.56,E2 -12131.56} C_VEL
LIN {X 0,Y 389.911,Z 418.566,A -85,B 0,C 180,E1 -12132.022,E2 -12132.022} C_VEL
LIN {X 0,Y 389.58,Z 431.243,A -85,B 0,C 180,E1 -12132.684,E2 -12132.684} C_VEL
LIN {X 0,Y 389.033,Z 442.862,A -85,B 0,C 180,E1 -12133.501,E2 -12133.501} C_VEL
LIN {X 0,Y 388.161,Z 454.044,A -85,B 0,C 180,E1 -12134.511,E2 -12134.511} C_VEL
LIN {X 0,Y 387.342,Z 464.378,A -85,B 0,C 180,E1 -12135.688,E2 -12135.688} C_VEL
LIN {X 0,Y 386.648,Z 472.801,A -85,B 0,C 180,E1 -12136.867,E2 -12136.867} C_VEL
LIN {X 0,Y 385.889,Z 480.556,A -85,B 0,C 180,E1 -12138.177,E2 -12138.177} C_VEL
LIN {X 0,Y 385.137,Z 488.23,A -85,B 0,C 180,E1 -12139.778,E2 -12139.778} C_VEL
LIN {X 0,Y 384.556,Z 493.985,A -85,B 0,C 180,E1 -12141.274,E2 -12141.274} C_VEL
LIN {X 0,Y 384.192,Z 498.256,A -85,B 0,C 180,E1 -12142.643,E2 -12142.643} C_VEL
LIN {X 0,Y 383.63,Z 502.152,A -85,B 0,C 180,E1 -12144.217,E2 -12144.217} C_VEL
LIN {X 0,Y 383.244,Z 505.022,A -85,B 0,C 180,E1 -12145.794,E2 -12145.794} C_VEL
LIN {X 0,Y 383.261,Z 506.371,A -85,B 0,C 180,E1 -12146.847,E2 -12146.847} C_VEL
LIN {X 0,Y 383.092,Z 507.353,A -85,B 0,C 180,E1 -12147.897,E2 -12147.897} C_VEL
LIN {X 0,Y 383.16,Z 507.935,A -85,B 0,C 180,E1 -12148.949,E2 -12148.949} C_VEL
LIN {X 0,Y 383.142,Z 508.164,A -85,B 0,C 180,E1 -12150,E2 -12150} C_VEL
LIN {X 0,Y 383.16,Z 507.979,A -85,B 0,C 180,E1 -12151.051,E2 -12151.051} C_VEL
LIN {X 0,Y 383.092,Z 507.425,A -85,B 0,C 180,E1 -12152.103,E2 -12152.103} C_VEL
LIN {X 0,Y 383.258,Z 506.471,A -85,B 0,C 180,E1 -12153.154,E2 -12153.154} C_VEL
LIN {X 0,Y 383.235,Z 505.169,A -85,B 0,C 180,E1 -12154.207,E2 -12154.207} C_VEL
LIN {X 0,Y 383.625,Z 502.352,A -85,B 0,C 180,E1 -12155.783,E2 -12155.783} C_VEL
LIN {X 0,Y 384.168,Z 498.526,A -85,B 0,C 180,E1 -12157.357,E2 -12157.357} C_VEL
LIN {X 0,Y 384.576,Z 493.45,A -85,B 0,C 180,E1 -12158.989,E2 -12158.989} C_VEL
LIN {X 0,Y 385.404,Z 486.215,A -85,B 0,C 180,E1 -12160.772,E2 -12160.772} C_VEL
LIN {X 0,Y 386.242,Z 478.187,A -85,B 0,C 180,E1 -12162.345,E2 -12162.345} C_VEL
LIN {X 0,Y 386.942,Z 469.966,A -85,B 0,C 180,E1 -12163.657,E2 -12163.657} C_VEL
LIN {X 0,Y 387.68,Z 460.935,A -85,B 0,C 180,E1 -12164.836,E2 -12164.836} C_VEL
LIN {X 0,Y 388.183,Z 454.98,A -85,B 0,C 180,E1 -12165.49,E2 -12165.49} C_VEL
LIN {X 0,Y 387.963,Z 450.203,A -85,B 0,C 180,E1 -12165.996,E2 -12165.996} C_VEL
LIN {X 0,Y 385.891,Z 442.269,A -85,B 0,C 180,E1 -12166.826,E2 -12166.826} C_VEL
LIN {X 0,Y 383.6,Z 434.038,A -85,B 0,C 180,E1 -12167.572,E2 -12167.572} C_VEL
LIN {X 0,Y 383.092,Z 428.709,A -85,B 0,C 180,E1 -12167.939,E2 -12167.939} C_VEL
LIN {X 0,Y 383.386,Z 416.334,A -85,B 0,C 180,E1 -12168.538,E2 -12168.538} C_VEL
LIN {X 0,Y 383.493,Z 404.619,A -85,B 0,C 180,E1 -12168.913,E2 -12168.913} C_VEL
LIN {X 0,Y 383.933,Z 358.314,A -85,B 0,C 180,E1 -12169.808,E2 -12169.808} C_VEL
LIN {X 0,Y 384.056,Z 344.68,A -85,B 0,C 180,E1 -12170.068,E2 -12170.068} C_VEL
LIN {X 0,Y 376.684,Z 326.991,A -85,B 0,C 180,E1 -12170.855,E2 -12170.855} C_VEL
LIN {X 0,Y 376.077,Z 325.22,A -85,B 0,C 180,E1 -12170.994,E2 -12170.994} C_VEL
LIN {X 0,Y 375.973,Z 324.696,A -85,B 0,C 180,E1 -12171.183,E2 -12171.183} C_VEL
LIN {X 0,Y 375.967,Z 324.652,A -85,B 0,C 180,E1 -12174.283,E2 -12174.283} C_VEL
LIN {X 0,Y 375.915,Z 324.625,A -85,B 0,C 180,E1 -12177.865,E2 -12177.865} C_VEL
LIN {X 0,Y 375.951,Z 324.658,A -85,B 0,C 180,E1 -12180.692,E2 -12180.692} C_VEL
LIN {X 0,Y 375.956,Z 324.651,A -85,B 0,C 180,E1 -12184.111,E2 -12184.111} C_VEL
LIN {X 0,Y 375.946,Z 324.642,A -85,B 0,C 180,E1 -12186.741,E2 -12186.741} C_VEL
LIN {X 0,Y 375.936,Z 324.655,A -85,B 0,C 180,E1 -12189.961,E2 -12189.961} C_VEL
LIN {X 0,Y 375.922,Z 324.639,A -85,B 0,C 180,E1 -12193.766,E2 -12193.766} C_VEL
LIN {X 0,Y 375.93,Z 324.66,A -85,B 0,C 180,E1 -12196.81,E2 -12196.81} C_VEL
LIN {X 0,Y 375.93,Z 324.629,A -85,B 0,C 180,E1 -12200.533,E2 -12200.533} C_VEL
LIN {X 0,Y 375.957,Z 324.647,A -85,B 0,C 180,E1 -12203.496,E2 -12203.496} C_VEL
LIN {X 0,Y 375.954,Z 324.653,A -85,B 0,C 180,E1 -12205.888,E2 -12205.888} C_VEL
LIN {X 0,Y 375.955,Z 324.618,A -85,B 0,C 180,E1 -12209.686,E2 -12209.686} C_VEL
LIN {X 0,Y 375.911,Z 324.632,A -85,B 0,C 180,E1 -12212.134,E2 -12212.134} C_VEL
LIN {X 0,Y 375.93,Z 324.654,A -85,B 0,C 180,E1 -12214.533,E2 -12214.533} C_VEL
LIN {X 0,Y 375.964,Z 324.65,A -85,B 0,C 180,E1 -12216.886,E2 -12216.886} C_VEL
LIN {X 0,Y 375.978,Z 324.644,A -85,B 0,C 180,E1 -12220.338,E2 -12220.338} C_VEL
LIN {X 0,Y 376.014,Z 324.643,A -85,B 0,C 180,E1 -12223.718,E2 -12223.718} C_VEL
LIN {X 0,Y 376.097,Z 324.633,A -85,B 0,C 180,E1 -12227.042,E2 -12227.042} C_VEL
LIN {X 0,Y 376.102,Z 324.632,A -85,B 0,C 180,E1 -12230.318,E2 -12230.318} C_VEL
LIN {X 0,Y 376.182,Z 324.617,A -85,B 0,C 180,E1 -12233.564,E2 -12233.564} C_VEL
LIN {X 0,Y 376.334,Z 324.603,A -85,B 0,C 180,E1 -12237.859,E2 -12237.859} C_VEL
LIN {X 0,Y 376.329,Z 324.607,A -85,B 0,C 180,E1 -12242.14,E2 -12242.14} C_VEL
LIN {X 0,Y 376.211,Z 324.61,A -85,B 0,C 180,E1 -12246.436,E2 -12246.436} C_VEL
LIN {X 0,Y 376.101,Z 324.634,A -85,B 0,C 180,E1 -12249.682,E2 -12249.682} C_VEL
LIN {X 0,Y 376.083,Z 324.626,A -85,B 0,C 180,E1 -12253.658,E2 -12253.658} C_VEL
LIN {X 0,Y 376.026,Z 324.642,A -85,B 0,C 180,E1 -12257.4,E2 -12257.4} C_VEL
LIN {X 0,Y 375.973,Z 324.627,A -85,B 0,C 180,E1 -12260.832,E2 -12260.832} C_VEL
LIN {X 0,Y 375.953,Z 324.657,A -85,B 0,C 180,E1 -12264.284,E2 -12264.284} C_VEL
LIN {X 0,Y 375.924,Z 324.643,A -85,B 0,C 180,E1 -12267.865,E2 -12267.865} C_VEL
LIN {X 0,Y 375.952,Z 324.654,A -85,B 0,C 180,E1 -12271.563,E2 -12271.563} C_VEL
LIN {X 0,Y 375.943,Z 324.646,A -85,B 0,C 180,E1 -12275.417,E2 -12275.417} C_VEL
LIN {X 0,Y 375.929,Z 324.652,A -85,B 0,C 180,E1 -12278.263,E2 -12278.263} C_VEL
LIN {X 0,Y 375.911,Z 324.66,A -85,B 0,C 180,E1 -12281.598,E2 -12281.598} C_VEL
LIN {X 0,Y 375.915,Z 324.628,A -85,B 0,C 180,E1 -12284.731,E2 -12284.731} C_VEL
LIN {X 0,Y 375.904,Z 324.661,A -85,B 0,C 180,E1 -12287.697,E2 -12287.697} C_VEL
LIN {X 0,Y 375.931,Z 324.639,A -85,B 0,C 180,E1 -12290.534,E2 -12290.534} C_VEL
LIN {X 0,Y 375.955,Z 324.646,A -85,B 0,C 180,E1 -12293.498,E2 -12293.498} C_VEL
LIN {X 0,Y 376.013,Z 324.853,A -85,B 0,C 180,E1 -12295.773,E2 -12295.773} C_VEL
LIN {X 0,Y 379.228,Z 338.207,A -85,B 0,C 180,E1 -12298.484,E2 -12298.484} C_VEL
LIN {X 0,Y 381.515,Z 349.01,A -85,B 0,C 180,E1 -12300.557,E2 -12300.557} C_VEL
LIN {X 0,Y 380.557,Z 362.147,A -85,B 0,C 180,E1 -12302.802,E2 -12302.802} C_VEL
LIN {X 0,Y 378.711,Z 383.926,A -85,B 0,C 180,E1 -12306.485,E2 -12306.485} C_VEL
LIN {X 0,Y 377.8,Z 396.844,A -85,B 0,C 180,E1 -12308.659,E2 -12308.659} C_VEL
LIN {X 0,Y 381.231,Z 425.836,A -85,B 0,C 180,E1 -12309.454,E2 -12309.454} C_VEL
LIN {X 0,Y 382.876,Z 444.813,A -85,B 0,C 180,E1 -12309.911,E2 -12309.911} C_VEL
LIN {X 0,Y 381.896,Z 507.702,A -85,B 0,C 180,E1 -12311.109,E2 -12311.109} C_VEL
LIN {X 0,Y 381.288,Z 520.983,A -85,B 0,C 180,E1 -12311.565,E2 -12311.565} C_VEL
LIN {X 0,Y 380.397,Z 533.181,A -85,B 0,C 180,E1 -12312.182,E2 -12312.182} C_VEL
LIN {X 0,Y 379.297,Z 545.523,A -85,B 0,C 180,E1 -12313.033,E2 -12313.033} C_VEL
LIN {X 0,Y 378.176,Z 557.226,A -85,B 0,C 180,E1 -12314.091,E2 -12314.091} C_VEL
LIN {X 0,Y 377.175,Z 567.803,A -85,B 0,C 180,E1 -12315.293,E2 -12315.293} C_VEL
LIN {X 0,Y 376.484,Z 576.85,A -85,B 0,C 180,E1 -12316.559,E2 -12316.559} C_VEL
LIN {X 0,Y 375.68,Z 585.947,A -85,B 0,C 180,E1 -12318.125,E2 -12318.125} C_VEL
LIN {X 0,Y 375.198,Z 593.576,A -85,B 0,C 180,E1 -12319.75,E2 -12319.75} C_VEL
LIN {X 0,Y 375.034,Z 599.746,A -85,B 0,C 180,E1 -12321.378,E2 -12321.378} C_VEL
LIN {X 0,Y 375.086,Z 605.305,A -85,B 0,C 180,E1 -12323.249,E2 -12323.249} C_VEL
LIN {X 0,Y 375.167,Z 608.412,A -85,B 0,C 180,E1 -12324.626,E2 -12324.626} C_VEL
LIN {X 0,Y 375.336,Z 610.369,A -85,B 0,C 180,E1 -12325.705,E2 -12325.705} C_VEL
LIN {X 0,Y 375.399,Z 611.829,A -85,B 0,C 180,E1 -12326.78,E2 -12326.78} C_VEL
LIN {X 0,Y 375.76,Z 613.545,A -85,B 0,C 180,E1 -12328.928,E2 -12328.928} C_VEL
LIN {X 0,Y 375.807,Z 613.775,A -85,B 0,C 180,E1 -12330,E2 -12330} C_VEL
LIN {X 0,Y 375.761,Z 613.542,A -85,B 0,C 180,E1 -12331.072,E2 -12331.072} C_VEL
LIN {X 0,Y 375.402,Z 611.824,A -85,B 0,C 180,E1 -12333.22,E2 -12333.22} C_VEL
LIN {X 0,Y 375.35,Z 610.362,A -85,B 0,C 180,E1 -12334.295,E2 -12334.295} C_VEL
LIN {X 0,Y 375.161,Z 607.283,A -85,B 0,C 180,E1 -12335.914,E2 -12335.914} C_VEL
LIN {X 0,Y 375.06,Z 603.139,A -85,B 0,C 180,E1 -12337.537,E2 -12337.537} C_VEL
LIN {X 0,Y 375.087,Z 596.796,A -85,B 0,C 180,E1 -12339.436,E2 -12339.436} C_VEL
LIN {X 0,Y 375.416,Z 589.921,A -85,B 0,C 180,E1 -12341.063,E2 -12341.063} C_VEL
LIN {X 0,Y 376.018,Z 581.438,A -85,B 0,C 180,E1 -12342.686,E2 -12342.686} C_VEL
LIN {X 0,Y 376.672,Z 572.762,A -85,B 0,C 180,E1 -12344.037,E2 -12344.037} C_VEL
LIN {X 0,Y 377.553,Z 563.296,A -85,B 0,C 180,E1 -12345.244,E2 -12345.244} C_VEL
LIN {X 0,Y 378.435,Z 554.488,A -85,B 0,C 180,E1 -12346.174,E2 -12346.174} C_VEL
LIN {X 0,Y 379.612,Z 541.908,A -85,B 0,C 180,E1 -12347.23,E2 -12347.23} C_VEL
LIN {X 0,Y 380.694,Z 529.595,A -85,B 0,C 180,E1 -12348.012,E2 -12348.012} C_VEL
LIN {X 0,Y 381.553,Z 516.657,A -85,B 0,C 180,E1 -12348.595,E2 -12348.595} C_VEL
LIN {X 0,Y 381.983,Z 502.911,A -85,B 0,C 180,E1 -12348.991,E2 -12348.991} C_VEL
LIN {X 0,Y 382.808,Z 443.113,A -85,B 0,C 180,E1 -12350.115,E2 -12350.115} C_VEL
LIN {X 0,Y 379.321,Z 409.492,A -85,B 0,C 180,E1 -12350.959,E2 -12350.959} C_VEL
LIN {X 0,Y 377.783,Z 397.136,A -85,B 0,C 180,E1 -12351.306,E2 -12351.306} C_VEL
LIN {X 0,Y 378.891,Z 382.199,A -85,B 0,C 180,E1 -12353.793,E2 -12353.793} C_VEL
LIN {X 0,Y 380.814,Z 358.86,A -85,B 0,C 180,E1 -12357.744,E2 -12357.744} C_VEL
LIN {X 0,Y 381.525,Z 348.931,A -85,B 0,C 180,E1 -12359.439,E2 -12359.439} C_VEL
LIN {X 0,Y 378.725,Z 335.911,A -85,B 0,C 180,E1 -12361.952,E2 -12361.952} C_VEL
LIN {X 0,Y 375.989,Z 324.768,A -85,B 0,C 180,E1 -12364.246,E2 -12364.246} C_VEL
LIN {X 0,Y 375.945,Z 324.651,A -85,B 0,C 180,E1 -12366.741,E2 -12366.741} C_VEL
LIN {X 0,Y 375.935,Z 324.64,A -85,B 0,C 180,E1 -12369.961,E2 -12369.961} C_VEL
LIN {X 0,Y 375.921,Z 324.638,A -85,B 0,C 180,E1 -12373.766,E2 -12373.766} C_VEL
LIN {X 0,Y 375.929,Z 324.65,A -85,B 0,C 180,E1 -12376.81,E2 -12376.81} C_VEL
LIN {X 0,Y 375.929,Z 324.643,A -85,B 0,C 180,E1 -12380.533,E2 -12380.533} C_VEL
LIN {X 0,Y 375.952,Z 324.604,A -85,B 0,C 180,E1 -12383.497,E2 -12383.497} C_VEL
LIN {X 0,Y 375.952,Z 324.639,A -85,B 0,C 180,E1 -12385.888,E2 -12385.888} C_VEL
LIN {X 0,Y 375.957,Z 324.649,A -85,B 0,C 180,E1 -12389.687,E2 -12389.687} C_VEL
LIN {X 0,Y 375.927,Z 324.643,A -85,B 0,C 180,E1 -12392.136,E2 -12392.136} C_VEL
LIN {X 0,Y 375.953,Z 324.657,A -85,B 0,C 180,E1 -12395.716,E2 -12395.716} C_VEL
LIN {X 0,Y 375.974,Z 324.627,A -85,B 0,C 180,E1 -12399.197,E2 -12399.197} C_VEL
LIN {X 0,Y 376.044,Z 324.64,A -85,B 0,C 180,E1 -12402.601,E2 -12402.601} C_VEL
LIN {X 0,Y 376.083,Z 324.625,A -85,B 0,C 180,E1 -12406.342,E2 -12406.342} C_VEL
LIN {X 0,Y 376.105,Z 324.634,A -85,B 0,C 180,E1 -12410.318,E2 -12410.318} C_VEL
LIN {X 0,Y 376.211,Z 324.611,A -85,B 0,C 180,E1 -12413.564,E2 -12413.564} C_VEL
LIN {X 0,Y 376.33,Z 324.608,A -85,B 0,C 180,E1 -12417.86,E2 -12417.86} C_VEL
LIN {X 0,Y 376.334,Z 324.602,A -85,B 0,C 180,E1 -12422.141,E2 -12422.141} C_VEL
LIN {X 0,Y 376.181,Z 324.616,A -85,B 0,C 180,E1 -12426.491,E2 -12426.491} C_VEL
LIN {X 0,Y 376.106,Z 324.631,A -85,B 0,C 180,E1 -12429.682,E2 -12429.682} C_VEL
LIN {X 0,Y 376.083,Z 324.627,A -85,B 0,C 180,E1 -12433.658,E2 -12433.658} C_VEL
LIN {X 0,Y 376.026,Z 324.645,A -85,B 0,C 180,E1 -12437.4,E2 -12437.4} C_VEL
LIN {X 0,Y 375.973,Z 324.64,A -85,B 0,C 180,E1 -12440.833,E2 -12440.833} C_VEL
LIN {X 0,Y 375.93,Z 324.655,A -85,B 0,C 180,E1 -12444.286,E2 -12444.286} C_VEL
LIN {X 0,Y 375.906,Z 324.649,A -85,B 0,C 180,E1 -12446.661,E2 -12446.661} C_VEL
LIN {X 0,Y 375.907,Z 324.621,A -85,B 0,C 180,E1 -12449.085,E2 -12449.085} C_VEL
LIN {X 0,Y 375.933,Z 324.633,A -85,B 0,C 180,E1 -12451.564,E2 -12451.564} C_VEL
LIN {X 0,Y 375.951,Z 324.656,A -85,B 0,C 180,E1 -12455.416,E2 -12455.416} C_VEL
LIN {X 0,Y 375.93,Z 324.633,A -85,B 0,C 180,E1 -12458.263,E2 -12458.263} C_VEL
LIN {X 0,Y 375.909,Z 324.652,A -85,B 0,C 180,E1 -12461.598,E2 -12461.598} C_VEL
LIN {X 0,Y 375.918,Z 324.656,A -85,B 0,C 180,E1 -12464.731,E2 -12464.731} C_VEL
LIN {X 0,Y 375.904,Z 324.644,A -85,B 0,C 180,E1 -12467.697,E2 -12467.697} C_VEL
LIN {X 0,Y 375.932,Z 324.656,A -85,B 0,C 180,E1 -12470.534,E2 -12470.534} C_VEL
LIN {X 0,Y 375.956,Z 324.642,A -85,B 0,C 180,E1 -12473.498,E2 -12473.498} C_VEL
LIN {X 0,Y 375.956,Z 324.652,A -85,B 0,C 180,E1 -12475.889,E2 -12475.889} C_VEL
LIN {X 0,Y 375.959,Z 324.654,A -85,B 0,C 180,E1 -12479.688,E2 -12479.688} C_VEL
LIN {X 0,Y 375.915,Z 324.627,A -85,B 0,C 180,E1 -12482.135,E2 -12482.135} C_VEL
LIN {X 0,Y 375.967,Z 324.656,A -85,B 0,C 180,E1 -12485.717,E2 -12485.717} C_VEL
LIN {X 0,Y 376.018,Z 324.845,A -85,B 0,C 180,E1 -12489.006,E2 -12489.006} C_VEL
LIN {X 0,Y 376.196,Z 325.632,A -85,B 0,C 180,E1 -12489.166,E2 -12489.166} C_VEL
LIN {X 0,Y 384.085,Z 344.63,A -85,B 0,C 180,E1 -12490.035,E2 -12490.035} C_VEL
LIN {X 0,Y 383.463,Z 405.338,A -85,B 0,C 180,E1 -12491.204,E2 -12491.204} C_VEL
LIN {X 0,Y 383.271,Z 418.133,A -85,B 0,C 180,E1 -12491.634,E2 -12491.634} C_VEL
LIN {X 0,Y 382.879,Z 431.117,A -85,B 0,C 180,E1 -12492.302,E2 -12492.302} C_VEL
LIN {X 0,Y 382.318,Z 443.451,A -85,B 0,C 180,E1 -12493.169,E2 -12493.169} C_VEL
LIN {X 0,Y 381.391,Z 455.027,A -85,B 0,C 180,E1 -12494.229,E2 -12494.229} C_VEL
LIN {X 0,Y 380.534,Z 465.36,A -85,B 0,C 180,E1 -12495.426,E2 -12495.426} C_VEL
LIN {X 0,Y 379.806,Z 473.782,A -85,B 0,C 180,E1 -12496.627,E2 -12496.627} C_VEL
LIN {X 0,Y 379.013,Z 481.536,A -85,B 0,C 180,E1 -12497.959,E2 -12497.959} C_VEL
LIN {X 0,Y 378.223,Z 489.21,A -85,B 0,C 180,E1 -12499.589,E2 -12499.589} C_VEL
LIN {X 0,Y 377.611,Z 494.964,A -85,B 0,C 180,E1 -12501.112,E2 -12501.112} C_VEL
LIN {X 0,Y 377.223,Z 499.235,A -85,B 0,C 180,E1 -12502.507,E2 -12502.507} C_VEL
LIN {X 0,Y 376.638,Z 503.131,A -85,B 0,C 180,E1 -12504.11,E2 -12504.11} C_VEL
LIN {X 0,Y 376.231,Z 506.002,A -85,B 0,C 180,E1 -12505.715,E2 -12505.715} C_VEL
LIN {X 0,Y 376.243,Z 507.349,A -85,B 0,C 180,E1 -12506.788,E2 -12506.788} C_VEL
LIN {X 0,Y 376.07,Z 508.331,A -85,B 0,C 180,E1 -12507.858,E2 -12507.858} C_VEL
LIN {X 0,Y 376.135,Z 508.913,A -85,B 0,C 180,E1 -12508.929,E2 -12508.929} C_VEL
LIN {X 0,Y 376.117,Z 509.141,A -85,B 0,C 180,E1 -12510,E2 -12510} C_VEL
LIN {X 0,Y 376.135,Z 508.956,A -85,B 0,C 180,E1 -12511.071,E2 -12511.071} C_VEL
LIN {X 0,Y 376.069,Z 508.403,A -85,B 0,C 180,E1 -12512.142,E2 -12512.142} C_VEL
LIN {X 0,Y 376.239,Z 507.449,A -85,B 0,C 180,E1 -12513.212,E2 -12513.212} C_VEL
LIN {X 0,Y 376.222,Z 506.147,A -85,B 0,C 180,E1 -12514.285,E2 -12514.285} C_VEL
LIN {X 0,Y 376.634,Z 503.329,A -85,B 0,C 180,E1 -12515.891,E2 -12515.891} C_VEL
LIN {X 0,Y 377.199,Z 499.503,A -85,B 0,C 180,E1 -12517.494,E2 -12517.494} C_VEL
LIN {X 0,Y 377.636,Z 494.426,A -85,B 0,C 180,E1 -12519.155,E2 -12519.155} C_VEL
LIN {X 0,Y 378.505,Z 487.19,A -85,B 0,C 180,E1 -12520.971,E2 -12520.971} C_VEL
LIN {X 0,Y 379.379,Z 479.162,A -85,B 0,C 180,E1 -12522.572,E2 -12522.572} C_VEL
LIN {X 0,Y 380.114,Z 470.941,A -85,B 0,C 180,E1 -12523.908,E2 -12523.908} C_VEL
LIN {X 0,Y 380.867,Z 461.913,A -85,B 0,C 180,E1 -12525.108,E2 -12525.108} C_VEL
LIN {X 0,Y 381.802,Z 451.405,A -85,B 0,C 180,E1 -12526.227,E2 -12526.227} C_VEL
LIN {X 0,Y 382.511,Z 439.74,A -85,B 0,C 180,E1 -12527.219,E2 -12527.219} C_VEL
LIN {X 0,Y 383.092,Z 428.709,A -85,B 0,C 180,E1 -12527.939,E2 -12527.939} C_VEL
LIN {X 0,Y 382.62,Z 423.256,A -85,B 0,C 180,E1 -12528.273,E2 -12528.273} C_VEL
LIN {X 0,Y 380.076,Z 414.347,A -85,B 0,C 180,E1 -12528.805,E2 -12528.805} C_VEL
LIN {X 0,Y 377.452,Z 405.242,A -85,B 0,C 180,E1 -12529.237,E2 -12529.237} C_VEL
LIN {X 0,Y 376.774,Z 399.485,A -85,B 0,C 180,E1 -12529.399,E2 -12529.399} C_VEL
LIN {X 0,Y 377.42,Z 346.283,A -85,B 0,C 180,E1 -12530.424,E2 -12530.424} C_VEL
LIN {X 0,Y 369.705,Z 328.024,A -85,B 0,C 180,E1 -12531.268,E2 -12531.268} C_VEL
LIN {X 0,Y 368.997,Z 326.037,A -85,B 0,C 180,E1 -12531.428,E2 -12531.428} C_VEL
LIN {X 0,Y 368.92,Z 325.544,A -85,B 0,C 180,E1 -12531.674,E2 -12531.674} C_VEL
LIN {X 0,Y 368.922,Z 325.532,A -85,B 0,C 180,E1 -12534.777,E2 -12534.777} C_VEL
LIN {X 0,Y 368.892,Z 325.511,A -85,B 0,C 180,E1 -12538.791,E2 -12538.791} C_VEL
LIN {X 0,Y 368.888,Z 325.526,A -85,B 0,C 180,E1 -12542.238,E2 -12542.238} C_VEL
LIN {X 0,Y 368.921,Z 325.532,A -85,B 0,C 180,E1 -12544.999,E2 -12544.999} C_VEL
LIN {X 0,Y 368.874,Z 325.527,A -85,B 0,C 180,E1 -12548.633,E2 -12548.633} C_VEL
LIN {X 0,Y 368.855,Z 325.527,A -85,B 0,C 180,E1 -12552.005,E2 -12552.005} C_VEL
LIN {X 0,Y 368.87,Z 325.533,A -85,B 0,C 180,E1 -12555.174,E2 -12555.174} C_VEL
LIN {X 0,Y 368.857,Z 325.536,A -85,B 0,C 180,E1 -12558.174,E2 -12558.174} C_VEL
LIN {X 0,Y 368.872,Z 325.508,A -85,B 0,C 180,E1 -12561.366,E2 -12561.366} C_VEL
LIN {X 0,Y 368.931,Z 325.528,A -85,B 0,C 180,E1 -12565.146,E2 -12565.146} C_VEL
LIN {X 0,Y 368.891,Z 325.503,A -85,B 0,C 180,E1 -12569.043,E2 -12569.043} C_VEL
LIN {X 0,Y 368.901,Z 325.499,A -85,B 0,C 180,E1 -12571.557,E2 -12571.557} C_VEL
LIN {X 0,Y 368.88,Z 325.534,A -85,B 0,C 180,E1 -12575.219,E2 -12575.219} C_VEL
LIN {X 0,Y 368.89,Z 325.529,A -85,B 0,C 180,E1 -12577.602,E2 -12577.602} C_VEL
LIN {X 0,Y 368.942,Z 325.526,A -85,B 0,C 180,E1 -12581.105,E2 -12581.105} C_VEL
LIN {X 0,Y 368.985,Z 325.511,A -85,B 0,C 180,E1 -12584.535,E2 -12584.535} C_VEL
LIN {X 0,Y 369.051,Z 325.509,A -85,B 0,C 180,E1 -12586.79,E2 -12586.79} C_VEL
LIN {X 0,Y 369.053,Z 325.513,A -85,B 0,C 180,E1 -12590.131,E2 -12590.131} C_VEL
LIN {X 0,Y 369.144,Z 325.494,A -85,B 0,C 180,E1 -12593.441,E2 -12593.441} C_VEL
LIN {X 0,Y 369.298,Z 325.479,A -85,B 0,C 180,E1 -12597.819,E2 -12597.819} C_VEL
LIN {X 0,Y 369.293,Z 325.484,A -85,B 0,C 180,E1 -12602.181,E2 -12602.181} C_VEL
LIN {X 0,Y 369.171,Z 325.487,A -85,B 0,C 180,E1 -12606.559,E2 -12606.559} C_VEL
LIN {X 0,Y 369.052,Z 325.513,A -85,B 0,C 180,E1 -12609.869,E2 -12609.869} C_VEL
LIN {X 0,Y 369.031,Z 325.505,A -85,B 0,C 180,E1 -12613.772,E2 -12613.772} C_VEL
LIN {X 0,Y 368.985,Z 325.52,A -85,B 0,C 180,E1 -12617.743,E2 -12617.743} C_VEL
LIN {X 0,Y 368.904,Z 325.509,A -85,B 0,C 180,E1 -12621.221,E2 -12621.221} C_VEL
LIN {X 0,Y 368.913,Z 325.529,A -85,B 0,C 180,E1 -12623.878,E2 -12623.878} C_VEL
LIN {X 0,Y 368.862,Z 325.527,A -85,B 0,C 180,E1 -12627.212,E2 -12627.212} C_VEL
LIN {X 0,Y 368.89,Z 325.523,A -85,B 0,C 180,E1 -12629.693,E2 -12629.693} C_VEL
LIN {X 0,Y 368.891,Z 325.529,A -85,B 0,C 180,E1 -12633.043,E2 -12633.043} C_VEL
LIN {X 0,Y 368.906,Z 325.53,A -85,B 0,C 180,E1 -12636.198,E2 -12636.198} C_VEL
LIN {X 0,Y 368.868,Z 325.527,A -85,B 0,C 180,E1 -12638.958,E2 -12638.958} C_VEL
LIN {X 0,Y 368.86,Z 325.538,A -85,B 0,C 180,E1 -12642.007,E2 -12642.007} C_VEL
LIN {X 0,Y 368.868,Z 325.505,A -85,B 0,C 180,E1 -12645.175,E2 -12645.175} C_VEL
LIN {X 0,Y 368.857,Z 325.539,A -85,B 0,C 180,E1 -12648.175,E2 -12648.175} C_VEL
LIN {X 0,Y 368.873,Z 325.524,A -85,B 0,C 180,E1 -12651.367,E2 -12651.367} C_VEL
LIN {X 0,Y 368.928,Z 325.536,A -85,B 0,C 180,E1 -12655.146,E2 -12655.146} C_VEL
LIN {X 0,Y 368.981,Z 325.825,A -85,B 0,C 180,E1 -12655.401,E2 -12655.401} C_VEL
LIN {X 0,Y 372.22,Z 339.153,A -85,B 0,C 180,E1 -12658.175,E2 -12658.175} C_VEL
LIN {X 0,Y 374.686,Z 351.271,A -85,B 0,C 180,E1 -12660.544,E2 -12660.544} C_VEL
LIN {X 0,Y 373.162,Z 367.927,A -85,B 0,C 180,E1 -12663.43,E2 -12663.43} C_VEL
LIN {X 0,Y 371.608,Z 386.247,A -85,B 0,C 180,E1 -12666.6,E2 -12666.6} C_VEL
LIN {X 0,Y 370.939,Z 395.839,A -85,B 0,C 180,E1 -12668.245,E2 -12668.245} C_VEL
LIN {X 0,Y 374.583,Z 427.065,A -85,B 0,C 180,E1 -12669.116,E2 -12669.116} C_VEL
LIN {X 0,Y 376.131,Z 445.867,A -85,B 0,C 180,E1 -12669.575,E2 -12669.575} C_VEL
LIN {X 0,Y 375.206,Z 506.73,A -85,B 0,C 180,E1 -12670.759,E2 -12670.759} C_VEL
LIN {X 0,Y 374.563,Z 520.005,A -85,B 0,C 180,E1 -12671.222,E2 -12671.222} C_VEL
LIN {X 0,Y 373.673,Z 532.204,A -85,B 0,C 180,E1 -12671.85,E2 -12671.85} C_VEL
LIN {X 0,Y 372.475,Z 544.534,A -85,B 0,C 180,E1 -12672.712,E2 -12672.712} C_VEL
LIN {X 0,Y 371.316,Z 556.236,A -85,B 0,C 180,E1 -12673.789,E2 -12673.789} C_VEL
LIN {X 0,Y 370.339,Z 565.72,A -85,B 0,C 180,E1 -12674.875,E2 -12674.875} C_VEL
LIN {X 0,Y 369.498,Z 574.458,A -85,B 0,C 180,E1 -12676.087,E2 -12676.087} C_VEL
LIN {X 0,Y 369.079,Z 580.501,A -85,B 0,C 180,E1 -12677.071,E2 -12677.071} C_VEL
LIN {X 0,Y 368.393,Z 588.968,A -85,B 0,C 180,E1 -12678.724,E2 -12678.724} C_VEL
LIN {X 0,Y 368.033,Z 595.835,A -85,B 0,C 180,E1 -12680.381,E2 -12680.381} C_VEL
LIN {X 0,Y 367.977,Z 602.17,A -85,B 0,C 180,E1 -12682.317,E2 -12682.317} C_VEL
LIN {X 0,Y 368.076,Z 606.309,A -85,B 0,C 180,E1 -12683.972,E2 -12683.972} C_VEL
LIN {X 0,Y 368.265,Z 609.383,A -85,B 0,C 180,E1 -12685.622,E2 -12685.622} C_VEL
LIN {X 0,Y 368.347,Z 610.847,A -85,B 0,C 180,E1 -12686.719,E2 -12686.719} C_VEL
LIN {X 0,Y 368.727,Z 612.567,A -85,B 0,C 180,E1 -12688.908,E2 -12688.908} C_VEL
LIN {X 0,Y 368.781,Z 612.797,A -85,B 0,C 180,E1 -12690,E2 -12690} C_VEL
LIN {X 0,Y 368.728,Z 612.563,A -85,B 0,C 180,E1 -12691.092,E2 -12691.092} C_VEL
LIN {X 0,Y 368.35,Z 610.841,A -85,B 0,C 180,E1 -12693.281,E2 -12693.281} C_VEL
LIN {X 0,Y 368.278,Z 609.375,A -85,B 0,C 180,E1 -12694.378,E2 -12694.378} C_VEL
LIN {X 0,Y 368.1,Z 606.295,A -85,B 0,C 180,E1 -12696.028,E2 -12696.028} C_VEL
LIN {X 0,Y 367.987,Z 602.145,A -85,B 0,C 180,E1 -12697.683,E2 -12697.683} C_VEL
LIN {X 0,Y 368.033,Z 595.799,A -85,B 0,C 180,E1 -12699.619,E2 -12699.619} C_VEL
LIN {X 0,Y 368.392,Z 588.923,A -85,B 0,C 180,E1 -12701.276,E2 -12701.276} C_VEL
LIN {X 0,Y 369.07,Z 580.444,A -85,B 0,C 180,E1 -12702.929,E2 -12702.929} C_VEL
LIN {X 0,Y 369.753,Z 571.766,A -85,B 0,C 180,E1 -12704.305,E2 -12704.305} C_VEL
LIN {X 0,Y 370.593,Z 562.288,A -85,B 0,C 180,E1 -12705.537,E2 -12705.537} C_VEL
LIN {X 0,Y 371.893,Z 550.614,A -85,B 0,C 180,E1 -12706.749,E2 -12706.749} C_VEL
LIN {X 0,Y 372.994,Z 539.132,A -85,B 0,C 180,E1 -12707.687,E2 -12707.687} C_VEL
LIN {X 0,Y 374.065,Z 527.366,A -85,B 0,C 180,E1 -12708.413,E2 -12708.413} C_VEL
LIN {X 0,Y 374.891,Z 513.817,A -85,B 0,C 180,E1 -12709.009,E2 -12709.009} C_VEL
LIN {X 0,Y 375.284,Z 500.344,A -85,B 0,C 180,E1 -12709.379,E2 -12709.379} C_VEL
LIN {X 0,Y 376.072,Z 443.099,A -85,B 0,C 180,E1 -12710.471,E2 -12710.471} C_VEL
LIN {X 0,Y 372.5,Z 409.147,A -85,B 0,C 180,E1 -12711.348,E2 -12711.348} C_VEL
LIN {X 0,Y 370.911,Z 395.983,A -85,B 0,C 180,E1 -12711.731,E2 -12711.731} C_VEL
LIN {X 0,Y 372.514,Z 375.169,A -85,B 0,C 180,E1 -12715.304,E2 -12715.304} C_VEL
LIN {X 0,Y 374.456,Z 354.361,A -85,B 0,C 180,E1 -12718.9,E2 -12718.9} C_VEL
LIN {X 0,Y 374.685,Z 351.188,A -85,B 0,C 180,E1 -12719.454,E2 -12719.454} C_VEL
LIN {X 0,Y 372.084,Z 338.558,A -85,B 0,C 180,E1 -12721.928,E2 -12721.928} C_VEL
LIN {X 0,Y 368.943,Z 325.644,A -85,B 0,C 180,E1 -12724.644,E2 -12724.644} C_VEL
LIN {X 0,Y 368.892,Z 325.538,A -85,B 0,C 180,E1 -12727.564,E2 -12727.564} C_VEL
LIN {X 0,Y 368.88,Z 325.522,A -85,B 0,C 180,E1 -12730.373,E2 -12730.373} C_VEL
LIN {X 0,Y 368.874,Z 325.518,A -85,B 0,C 180,E1 -12733.614,E2 -12733.614} C_VEL
LIN {X 0,Y 368.879,Z 325.524,A -85,B 0,C 180,E1 -12736.695,E2 -12736.695} C_VEL
LIN {X 0,Y 368.88,Z 325.531,A -85,B 0,C 180,E1 -12739.648,E2 -12739.648} C_VEL
LIN {X 0,Y 368.89,Z 325.481,A -85,B 0,C 180,E1 -12743.145,E2 -12743.145} C_VEL
LIN {X 0,Y 368.89,Z 325.529,A -85,B 0,C 180,E1 -12746.461,E2 -12746.461} C_VEL
LIN {X 0,Y 368.908,Z 325.53,A -85,B 0,C 180,E1 -12749.044,E2 -12749.044} C_VEL
LIN {X 0,Y 368.91,Z 325.514,A -85,B 0,C 180,E1 -12751.558,E2 -12751.558} C_VEL
LIN {X 0,Y 368.892,Z 325.533,A -85,B 0,C 180,E1 -12755.22,E2 -12755.22} C_VEL
LIN {X 0,Y 368.914,Z 325.518,A -85,B 0,C 180,E1 -12757.604,E2 -12757.604} C_VEL
LIN {X 0,Y 368.951,Z 325.513,A -85,B 0,C 180,E1 -12761.106,E2 -12761.106} C_VEL
LIN {X 0,Y 368.991,Z 325.519,A -85,B 0,C 180,E1 -12764.535,E2 -12764.535} C_VEL
